ABB RAPID module: P707.mod

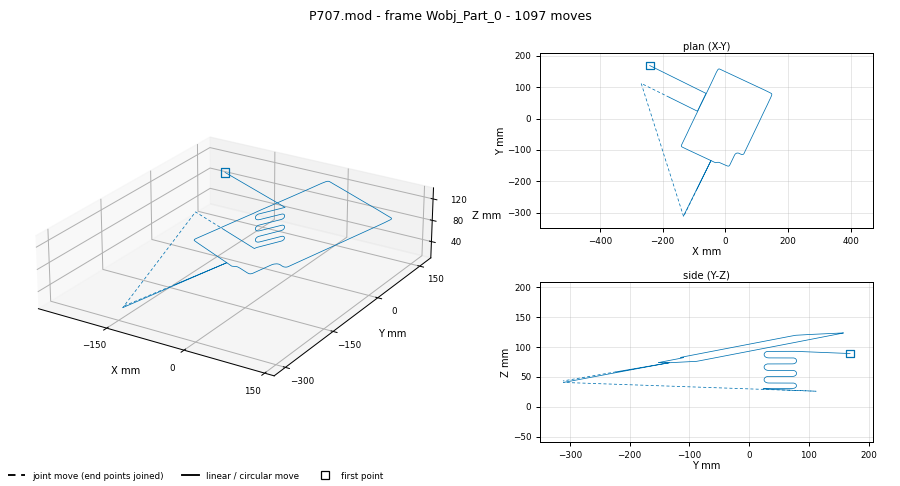
[picture p0: tool path of P707.mod in frame Wobj_Part_0, 1097 of 1107 moves have a stored position in this frame; points joined in program order, loops and branches not executed]
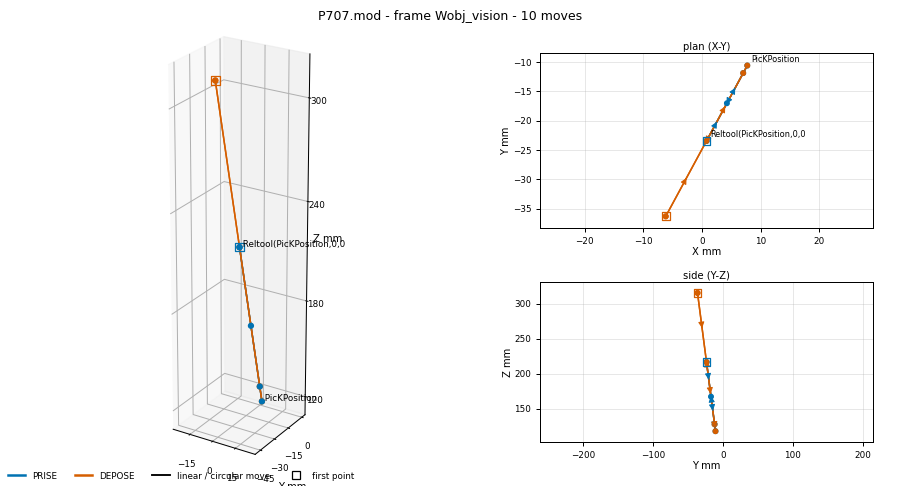
[picture p1: tool path of P707.mod in frame Wobj_vision, 10 of 1107 moves have a stored position in this frame; points joined in program order, loops and branches not executed]
MODULE P707

    ! Nom         :P707
    ! Description :
    ! Créé le     :30/05/2023 16:24:55

    LOCAL CONST SPEEDDATA VitesseLente :=[3,500,0,0];
	LOCAL CONST SPEEDDATA VitesseRapide :=[30,500,0,0];
	LOCAL CONST SPEEDDATA VitesseTronconnage :=[2,500,0,0];
	LOCAL CONST SPEEDDATA VitesseTronconnageApp :=[10,500,0,0];
    !
    !Point de prise
    LOCAL PERS Robtarget PicKPosition := [[7.7250060607796,-10.5869305006045,117.632375104374],[0.0368021435703274,-0.850900226645692,-0.520193892005484,-0.0633460436264631],[0,0,0,0],[8.999999E+09,8.999999E+09,8.999999E+09,8.999999E+09,8.999999E+09,8.999999E+09]];
	LOCAL PERS Pose Ref := [[0,0,0],[1,0,0,0]];
    !
    !Declaration des points de meulage

    !Tr_meulage_motif_1 : Meulage d'un motif
    LOCAL CONST Robtarget Tr_meulage_motif_1_0 := [[-61.692015625,80.0117578125,92.8283359375],[0.376363228761976,-0.369466106511504,0.595187364718739,-0.60629820802494],[0,0,0,0],[8.999999E+09,8.999999E+09,8.999999E+09,8.999999E+09,8.999999E+09,8.999999E+09]];
    LOCAL CONST Robtarget Tr_meulage_motif_1_1 := [[-62.12769921875,79.11165625,92.8283359375],[0.376363228761976,-0.369466106511504,0.595187364718739,-0.60629820802494],[0,0,0,0],[8.999999E+09,8.999999E+09,8.999999E+09,8.999999E+09,8.999999E+09,8.999999E+09]];
    LOCAL CONST Robtarget Tr_meulage_motif_1_2 := [[-62.5633828125,78.2115546875,92.82834375],[0.376363228761976,-0.369466106511504,0.595187364718739,-0.60629820802494],[0,0,0,0],[8.999999E+09,8.999999E+09,8.999999E+09,8.999999E+09,8.999999E+09,8.999999E+09]];
    LOCAL CONST Robtarget Tr_meulage_motif_1_3 := [[-62.99906640625,77.3114609375,92.82834375],[0.376363228761976,-0.369466106511504,0.595187364718739,-0.60629820802494],[0,0,0,0],[8.999999E+09,8.999999E+09,8.999999E+09,8.999999E+09,8.999999E+09,8.999999E+09]];
    LOCAL CONST Robtarget Tr_meulage_motif_1_4 := [[-63.43475,76.411359375,92.8283515625],[0.376363228761976,-0.369466106511504,0.595187364718739,-0.60629820802494],[0,0,0,0],[8.999999E+09,8.999999E+09,8.999999E+09,8.999999E+09,8.999999E+09,8.999999E+09]];
    LOCAL CONST Robtarget Tr_meulage_motif_1_5 := [[-63.8704375,75.5112578125,92.8283515625],[0.376363228761976,-0.369466106511504,0.595187364718739,-0.60629820802494],[0,0,0,0],[8.999999E+09,8.999999E+09,8.999999E+09,8.999999E+09,8.999999E+09,8.999999E+09]];
    LOCAL CONST Robtarget Tr_meulage_motif_1_6 := [[-64.30612109375,74.61115625,92.828359375],[0.376363228761976,-0.369466106511504,0.595187364718739,-0.60629820802494],[0,0,0,0],[8.999999E+09,8.999999E+09,8.999999E+09,8.999999E+09,8.999999E+09,8.999999E+09]];
    LOCAL CONST Robtarget Tr_meulage_motif_1_7 := [[-64.7418046875,73.7110625,92.828359375],[0.376363228761976,-0.369466106511504,0.595187364718739,-0.60629820802494],[0,0,0,0],[8.999999E+09,8.999999E+09,8.999999E+09,8.999999E+09,8.999999E+09,8.999999E+09]];
    LOCAL CONST Robtarget Tr_meulage_motif_1_8 := [[-65.17748828125,72.8109609375,92.828359375],[0.376363228761976,-0.369466106511504,0.595187364718739,-0.60629820802494],[0,0,0,0],[8.999999E+09,8.999999E+09,8.999999E+09,8.999999E+09,8.999999E+09,8.999999E+09]];
    LOCAL CONST Robtarget Tr_meulage_motif_1_9 := [[-65.613171875,71.910859375,92.8283671875],[0.376363228761976,-0.369466106511504,0.595187364718739,-0.60629820802494],[0,0,0,0],[8.999999E+09,8.999999E+09,8.999999E+09,8.999999E+09,8.999999E+09,8.999999E+09]];
    LOCAL CONST Robtarget Tr_meulage_motif_1_10 := [[-66.048859375,71.0107578125,92.8283671875],[0.376363228761976,-0.369466106511504,0.595187364718739,-0.60629820802494],[0,0,0,0],[8.999999E+09,8.999999E+09,8.999999E+09,8.999999E+09,8.999999E+09,8.999999E+09]];
    LOCAL CONST Robtarget Tr_meulage_motif_1_11 := [[-66.4845390625,70.1106640625,92.828375],[0.376363228761976,-0.369466106511504,0.595187364718739,-0.60629820802494],[0,0,0,0],[8.999999E+09,8.999999E+09,8.999999E+09,8.999999E+09,8.999999E+09,8.999999E+09]];
    LOCAL CONST Robtarget Tr_meulage_motif_1_12 := [[-66.9202265625,69.2105625,92.828375],[0.376363228761976,-0.369466106511504,0.595187364718739,-0.60629820802494],[0,0,0,0],[8.999999E+09,8.999999E+09,8.999999E+09,8.999999E+09,8.999999E+09,8.999999E+09]];
    LOCAL CONST Robtarget Tr_meulage_motif_1_13 := [[-67.35590625,68.3104609375,92.8283828125],[0.376363228761976,-0.369466106511504,0.595187364718739,-0.60629820802494],[0,0,0,0],[8.999999E+09,8.999999E+09,8.999999E+09,8.999999E+09,8.999999E+09,8.999999E+09]];
    LOCAL CONST Robtarget Tr_meulage_motif_1_14 := [[-67.79159375,67.410359375,92.8283828125],[0.376363228761976,-0.369466106511504,0.595187364718739,-0.60629820802494],[0,0,0,0],[8.999999E+09,8.999999E+09,8.999999E+09,8.999999E+09,8.999999E+09,8.999999E+09]];
    LOCAL CONST Robtarget Tr_meulage_motif_1_15 := [[-68.22728125,66.510265625,92.8283828125],[0.376363228761976,-0.369466106511504,0.595187364718739,-0.60629820802494],[0,0,0,0],[8.999999E+09,8.999999E+09,8.999999E+09,8.999999E+09,8.999999E+09,8.999999E+09]];
    LOCAL CONST Robtarget Tr_meulage_motif_1_16 := [[-68.6629609375,65.6101640625,92.828390625],[0.376363228761976,-0.369466106511504,0.595187364718739,-0.60629820802494],[0,0,0,0],[8.999999E+09,8.999999E+09,8.999999E+09,8.999999E+09,8.999999E+09,8.999999E+09]];
    LOCAL CONST Robtarget Tr_meulage_motif_1_17 := [[-69.0986484375,64.7100625,92.828390625],[0.376363228761976,-0.369466106511504,0.595187364718739,-0.60629820802494],[0,0,0,0],[8.999999E+09,8.999999E+09,8.999999E+09,8.999999E+09,8.999999E+09,8.999999E+09]];
    LOCAL CONST Robtarget Tr_meulage_motif_1_18 := [[-69.534328125,63.80996484375,92.8283984375],[0.376363228761976,-0.369466106511504,0.595187364718739,-0.60629820802494],[0,0,0,0],[8.999999E+09,8.999999E+09,8.999999E+09,8.999999E+09,8.999999E+09,8.999999E+09]];
    LOCAL CONST Robtarget Tr_meulage_motif_1_19 := [[-69.970015625,62.90986328125,92.8283984375],[0.376363228761976,-0.369466106511504,0.595187364718739,-0.60629820802494],[0,0,0,0],[8.999999E+09,8.999999E+09,8.999999E+09,8.999999E+09,8.999999E+09,8.999999E+09]];
    LOCAL CONST Robtarget Tr_meulage_motif_1_20 := [[-70.405703125,62.009765625,92.82840625],[0.376363228761976,-0.369466106511504,0.595187364718739,-0.60629820802494],[0,0,0,0],[8.999999E+09,8.999999E+09,8.999999E+09,8.999999E+09,8.999999E+09,8.999999E+09]];
    LOCAL CONST Robtarget Tr_meulage_motif_1_21 := [[-70.8413828125,61.1096640625,92.82840625],[0.376363228761976,-0.369466106511504,0.595187364718739,-0.60629820802494],[0,0,0,0],[8.999999E+09,8.999999E+09,8.999999E+09,8.999999E+09,8.999999E+09,8.999999E+09]];
    LOCAL CONST Robtarget Tr_meulage_motif_1_22 := [[-71.2770703125,60.20956640625,92.82840625],[0.376363228761976,-0.369466106511504,0.595187364718739,-0.60629820802494],[0,0,0,0],[8.999999E+09,8.999999E+09,8.999999E+09,8.999999E+09,8.999999E+09,8.999999E+09]];
    LOCAL CONST Robtarget Tr_meulage_motif_1_23 := [[-71.71275,59.30946484375,92.8284140625],[0.376363228761976,-0.369466106511504,0.595187364718739,-0.60629820802494],[0,0,0,0],[8.999999E+09,8.999999E+09,8.999999E+09,8.999999E+09,8.999999E+09,8.999999E+09]];
    LOCAL CONST Robtarget Tr_meulage_motif_1_24 := [[-72.1484375,58.4093671875,92.8284140625],[0.376363228761976,-0.369466106511504,0.595187364718739,-0.60629820802494],[0,0,0,0],[8.999999E+09,8.999999E+09,8.999999E+09,8.999999E+09,8.999999E+09,8.999999E+09]];
    LOCAL CONST Robtarget Tr_meulage_motif_1_25 := [[-72.5841171875,57.509265625,92.828421875],[0.376363228761976,-0.369466106511504,0.595187364718739,-0.60629820802494],[0,0,0,0],[8.999999E+09,8.999999E+09,8.999999E+09,8.999999E+09,8.999999E+09,8.999999E+09]];
    LOCAL CONST Robtarget Tr_meulage_motif_1_26 := [[-73.0198046875,56.60916796875,92.828421875],[0.376363228761976,-0.369466106511504,0.595187364718739,-0.60629820802494],[0,0,0,0],[8.999999E+09,8.999999E+09,8.999999E+09,8.999999E+09,8.999999E+09,8.999999E+09]];
    LOCAL CONST Robtarget Tr_meulage_motif_1_27 := [[-73.4554921875,55.70906640625,92.8284296875],[0.376363228761976,-0.369466106511504,0.595187364718739,-0.60629820802494],[0,0,0,0],[8.999999E+09,8.999999E+09,8.999999E+09,8.999999E+09,8.999999E+09,8.999999E+09]];
    LOCAL CONST Robtarget Tr_meulage_motif_1_28 := [[-73.891171875,54.80896875,92.8284296875],[0.376363228761976,-0.369466106511504,0.595187364718739,-0.60629820802494],[0,0,0,0],[8.999999E+09,8.999999E+09,8.999999E+09,8.999999E+09,8.999999E+09,8.999999E+09]];
    LOCAL CONST Robtarget Tr_meulage_motif_1_29 := [[-74.326859375,53.9088671875,92.8284296875],[0.376363228761976,-0.369466106511504,0.595187364718739,-0.60629820802494],[0,0,0,0],[8.999999E+09,8.999999E+09,8.999999E+09,8.999999E+09,8.999999E+09,8.999999E+09]];
    LOCAL CONST Robtarget Tr_meulage_motif_1_30 := [[-74.7625390625,53.00876953125,92.8284375],[0.376363228761976,-0.369466106511504,0.595187364718739,-0.60629820802494],[0,0,0,0],[8.999999E+09,8.999999E+09,8.999999E+09,8.999999E+09,8.999999E+09,8.999999E+09]];
    LOCAL CONST Robtarget Tr_meulage_motif_1_31 := [[-75.1982265625,52.10866796875,92.8284375],[0.376363228761976,-0.369466106511504,0.595187364718739,-0.60629820802494],[0,0,0,0],[8.999999E+09,8.999999E+09,8.999999E+09,8.999999E+09,8.999999E+09,8.999999E+09]];
    LOCAL CONST Robtarget Tr_meulage_motif_1_32 := [[-75.6339140625,51.2085703125,92.8284453125],[0.376363228761976,-0.369466106511504,0.595187364718739,-0.60629820802494],[0,0,0,0],[8.999999E+09,8.999999E+09,8.999999E+09,8.999999E+09,8.999999E+09,8.999999E+09]];
    LOCAL CONST Robtarget Tr_meulage_motif_1_33 := [[-76.06959375,50.30846875,92.8284453125],[0.376363228761976,-0.369466106511504,0.595187364718739,-0.60629820802494],[0,0,0,0],[8.999999E+09,8.999999E+09,8.999999E+09,8.999999E+09,8.999999E+09,8.999999E+09]];
    LOCAL CONST Robtarget Tr_meulage_motif_1_34 := [[-76.50528125,49.40837109375,92.828453125],[0.376363228761976,-0.369466106511504,0.595187364718739,-0.60629820802494],[0,0,0,0],[8.999999E+09,8.999999E+09,8.999999E+09,8.999999E+09,8.999999E+09,8.999999E+09]];
    LOCAL CONST Robtarget Tr_meulage_motif_1_35 := [[-76.9409609375,48.50826953125,92.828453125],[0.376363228761976,-0.369466106511504,0.595187364718739,-0.60629820802494],[0,0,0,0],[8.999999E+09,8.999999E+09,8.999999E+09,8.999999E+09,8.999999E+09,8.999999E+09]];
    LOCAL CONST Robtarget Tr_meulage_motif_1_36 := [[-77.3766484375,47.608171875,92.828453125],[0.376363228761976,-0.369466106511504,0.595187364718739,-0.60629820802494],[0,0,0,0],[8.999999E+09,8.999999E+09,8.999999E+09,8.999999E+09,8.999999E+09,8.999999E+09]];
    LOCAL CONST Robtarget Tr_meulage_motif_1_37 := [[-77.812328125,46.7080703125,92.8284609375],[0.376363228761976,-0.369466106511504,0.595187364718739,-0.60629820802494],[0,0,0,0],[8.999999E+09,8.999999E+09,8.999999E+09,8.999999E+09,8.999999E+09,8.999999E+09]];
    LOCAL CONST Robtarget Tr_meulage_motif_1_38 := [[-78.248015625,45.80797265625,92.8284609375],[0.376363228761976,-0.369466106511504,0.595187364718739,-0.60629820802494],[0,0,0,0],[8.999999E+09,8.999999E+09,8.999999E+09,8.999999E+09,8.999999E+09,8.999999E+09]];
    LOCAL CONST Robtarget Tr_meulage_motif_1_39 := [[-78.683703125,44.907875,92.82846875],[0.376363228761976,-0.369466106511504,0.595187364718739,-0.60629820802494],[0,0,0,0],[8.999999E+09,8.999999E+09,8.999999E+09,8.999999E+09,8.999999E+09,8.999999E+09]];
    LOCAL CONST Robtarget Tr_meulage_motif_1_40 := [[-79.1193828125,44.0077734375,92.82846875],[0.376363228761976,-0.369466106511504,0.595187364718739,-0.60629820802494],[0,0,0,0],[8.999999E+09,8.999999E+09,8.999999E+09,8.999999E+09,8.999999E+09,8.999999E+09]];
    LOCAL CONST Robtarget Tr_meulage_motif_1_41 := [[-79.5550703125,43.10767578125,92.8284765625],[0.376363228761976,-0.369466106511504,0.595187364718739,-0.60629820802494],[0,0,0,0],[8.999999E+09,8.999999E+09,8.999999E+09,8.999999E+09,8.999999E+09,8.999999E+09]];
    LOCAL CONST Robtarget Tr_meulage_motif_1_42 := [[-79.99075,42.20757421875,92.8284765625],[0.376363228761976,-0.369466106511504,0.595187364718739,-0.60629820802494],[0,0,0,0],[8.999999E+09,8.999999E+09,8.999999E+09,8.999999E+09,8.999999E+09,8.999999E+09]];
    LOCAL CONST Robtarget Tr_meulage_motif_1_43 := [[-80.4264375,41.3074765625,92.8284765625],[0.376363228761976,-0.369466106511504,0.595187364718739,-0.60629820802494],[0,0,0,0],[8.999999E+09,8.999999E+09,8.999999E+09,8.999999E+09,8.999999E+09,8.999999E+09]];
    LOCAL CONST Robtarget Tr_meulage_motif_1_44 := [[-80.862125,40.407375,92.828484375],[0.376363228761976,-0.369466106511504,0.595187364718739,-0.60629820802494],[0,0,0,0],[8.999999E+09,8.999999E+09,8.999999E+09,8.999999E+09,8.999999E+09,8.999999E+09]];
    LOCAL CONST Robtarget Tr_meulage_motif_1_45 := [[-81.2978046875,39.50727734375,92.828484375],[0.376363228761976,-0.369466106511504,0.595187364718739,-0.60629820802494],[0,0,0,0],[8.999999E+09,8.999999E+09,8.999999E+09,8.999999E+09,8.999999E+09,8.999999E+09]];
    LOCAL CONST Robtarget Tr_meulage_motif_1_46 := [[-81.7334921875,38.60717578125,92.8284921875],[0.376363228761976,-0.369466106511504,0.595187364718739,-0.60629820802494],[0,0,0,0],[8.999999E+09,8.999999E+09,8.999999E+09,8.999999E+09,8.999999E+09,8.999999E+09]];
    LOCAL CONST Robtarget Tr_meulage_motif_1_47 := [[-82.169171875,37.707078125,92.8284921875],[0.376363228761976,-0.369466106511504,0.595187364718739,-0.60629820802494],[0,0,0,0],[8.999999E+09,8.999999E+09,8.999999E+09,8.999999E+09,8.999999E+09,8.999999E+09]];
    LOCAL CONST Robtarget Tr_meulage_motif_1_48 := [[-82.604859375,36.8069765625,92.8285],[0.376363228761976,-0.369466106511504,0.595187364718739,-0.60629820802494],[0,0,0,0],[8.999999E+09,8.999999E+09,8.999999E+09,8.999999E+09,8.999999E+09,8.999999E+09]];
    LOCAL CONST Robtarget Tr_meulage_motif_1_49 := [[-83.0405390625,35.90687890625,92.8285],[0.376363228761976,-0.369466106511504,0.595187364718739,-0.60629820802494],[0,0,0,0],[8.999999E+09,8.999999E+09,8.999999E+09,8.999999E+09,8.999999E+09,8.999999E+09]];
    LOCAL CONST Robtarget Tr_meulage_motif_1_50 := [[-83.4762265625,35.00677734375,92.8285],[0.376363228761976,-0.369466106511504,0.595187364718739,-0.60629820802494],[0,0,0,0],[8.999999E+09,8.999999E+09,8.999999E+09,8.999999E+09,8.999999E+09,8.999999E+09]];
    LOCAL CONST Robtarget Tr_meulage_motif_1_51 := [[-83.9119140625,34.1066796875,92.8285078125],[0.376363228761976,-0.369466106511504,0.595187364718739,-0.60629820802494],[0,0,0,0],[8.999999E+09,8.999999E+09,8.999999E+09,8.999999E+09,8.999999E+09,8.999999E+09]];
    LOCAL CONST Robtarget Tr_meulage_motif_1_52 := [[-84.34759375,33.206578125,92.8285078125],[0.376363228761976,-0.369466106511504,0.595187364718739,-0.60629820802494],[0,0,0,0],[8.999999E+09,8.999999E+09,8.999999E+09,8.999999E+09,8.999999E+09,8.999999E+09]];
    LOCAL CONST Robtarget Tr_meulage_motif_1_53 := [[-84.78328125,32.306478515625,92.828515625],[0.376363228761976,-0.369466106511504,0.595187364718739,-0.60629820802494],[0,0,0,0],[8.999999E+09,8.999999E+09,8.999999E+09,8.999999E+09,8.999999E+09,8.999999E+09]];
    LOCAL CONST Robtarget Tr_meulage_motif_1_54 := [[-85.2189609375,31.40637890625,92.828515625],[0.376363228761976,-0.369466106511504,0.595187364718739,-0.60629820802494],[0,0,0,0],[8.999999E+09,8.999999E+09,8.999999E+09,8.999999E+09,8.999999E+09,8.999999E+09]];
    LOCAL CONST Robtarget Tr_meulage_motif_1_55 := [[-85.650984375,30.512767578125,92.7179296875],[0.376363228761976,-0.369466106511504,0.595187364718739,-0.60629820802494],[0,0,0,0],[8.999999E+09,8.999999E+09,8.999999E+09,8.999999E+09,8.999999E+09,8.999999E+09]];
    LOCAL CONST Robtarget Tr_meulage_motif_1_56 := [[-86.0625390625,29.660427734375,92.5067421875],[0.376363228761976,-0.369466106511504,0.595187364718739,-0.60629820802494],[0,0,0,0],[8.999999E+09,8.999999E+09,8.999999E+09,8.999999E+09,8.999999E+09,8.999999E+09]];
    LOCAL CONST Robtarget Tr_meulage_motif_1_57 := [[-86.4330078125,28.892388671875,92.23490625],[0.376363228761976,-0.369466106511504,0.595187364718739,-0.60629820802494],[0,0,0,0],[8.999999E+09,8.999999E+09,8.999999E+09,8.999999E+09,8.999999E+09,8.999999E+09]];
    LOCAL CONST Robtarget Tr_meulage_motif_1_58 := [[-86.7586796875,28.216853515625,91.9589765625],[0.376363228761976,-0.369466106511504,0.595187364718739,-0.60629820802494],[0,0,0,0],[8.999999E+09,8.999999E+09,8.999999E+09,8.999999E+09,8.999999E+09,8.999999E+09]];
    LOCAL CONST Robtarget Tr_meulage_motif_1_59 := [[-87.2360234375,27.22463671875,91.342859375],[0.376363228761976,-0.369466106511504,0.595187364718739,-0.60629820802494],[0,0,0,0],[8.999999E+09,8.999999E+09,8.999999E+09,8.999999E+09,8.999999E+09,8.999999E+09]];
    LOCAL CONST Robtarget Tr_meulage_motif_1_60 := [[-87.67884375,26.3014609375,90.4952109375],[0.376363228761976,-0.369466106511504,0.595187364718739,-0.60629820802494],[0,0,0,0],[8.999999E+09,8.999999E+09,8.999999E+09,8.999999E+09,8.999999E+09,8.999999E+09]];
    LOCAL CONST Robtarget Tr_meulage_motif_1_61 := [[-88.044203125,25.536572265625,89.4713515625],[0.376363228761976,-0.369466106511504,0.595187364718739,-0.60629820802494],[0,0,0,0],[8.999999E+09,8.999999E+09,8.999999E+09,8.999999E+09,8.999999E+09,8.999999E+09]];
    LOCAL CONST Robtarget Tr_meulage_motif_1_62 := [[-88.2525859375,25.095095703125,88.355171875],[0.376363228761976,-0.369466106511504,0.595187364718739,-0.60629820802494],[0,0,0,0],[8.999999E+09,8.999999E+09,8.999999E+09,8.999999E+09,8.999999E+09,8.999999E+09]];
    LOCAL CONST Robtarget Tr_meulage_motif_1_63 := [[-88.2616875,25.069435546875,87.6592109375],[0.376363228761976,-0.369466106511504,0.595187364718739,-0.60629820802494],[0,0,0,0],[8.999999E+09,8.999999E+09,8.999999E+09,8.999999E+09,8.999999E+09,8.999999E+09]];
    LOCAL CONST Robtarget Tr_meulage_motif_1_64 := [[-88.259140625,25.06819921875,86.99796875],[0.376363228761976,-0.369466106511504,0.595187364718739,-0.60629820802494],[0,0,0,0],[8.999999E+09,8.999999E+09,8.999999E+09,8.999999E+09,8.999999E+09,8.999999E+09]];
    LOCAL CONST Robtarget Tr_meulage_motif_1_65 := [[-88.2326796875,25.11635546875,86.3368828125],[0.376363228761976,-0.369466106511504,0.595187364718739,-0.60629820802494],[0,0,0,0],[8.999999E+09,8.999999E+09,8.999999E+09,8.999999E+09,8.999999E+09,8.999999E+09]];
    LOCAL CONST Robtarget Tr_meulage_motif_1_66 := [[-88.0113671875,25.5627421875,85.235140625],[0.376363228761976,-0.369466106511504,0.595187364718739,-0.60629820802494],[0,0,0,0],[8.999999E+09,8.999999E+09,8.999999E+09,8.999999E+09,8.999999E+09,8.999999E+09]];
    LOCAL CONST Robtarget Tr_meulage_motif_1_67 := [[-87.6342734375,26.33190625,84.2285234375],[0.376363228761976,-0.369466106511504,0.595187364718739,-0.60629820802494],[0,0,0,0],[8.999999E+09,8.999999E+09,8.999999E+09,8.999999E+09,8.999999E+09,8.999999E+09]];
    LOCAL CONST Robtarget Tr_meulage_motif_1_68 := [[-87.1851953125,27.251525390625,83.3996484375],[0.376363228761976,-0.369466106511504,0.595187364718739,-0.60629820802494],[0,0,0,0],[8.999999E+09,8.999999E+09,8.999999E+09,8.999999E+09,8.999999E+09,8.999999E+09]];
    LOCAL CONST Robtarget Tr_meulage_motif_1_69 := [[-86.8843125,27.86923828125,83.0038984375],[0.376363228761976,-0.369466106511504,0.595187364718739,-0.60629820802494],[0,0,0,0],[8.999999E+09,8.999999E+09,8.999999E+09,8.999999E+09,8.999999E+09,8.999999E+09]];
    LOCAL CONST Robtarget Tr_meulage_motif_1_70 := [[-86.37784375,28.91078125,82.5163671875],[0.376363228761976,-0.369466106511504,0.595187364718739,-0.60629820802494],[0,0,0,0],[8.999999E+09,8.999999E+09,8.999999E+09,8.999999E+09,8.999999E+09,8.999999E+09]];
    LOCAL CONST Robtarget Tr_meulage_motif_1_71 := [[-86.00865625,29.670900390625,82.2522734375],[0.376363228761976,-0.369466106511504,0.595187364718739,-0.60629820802494],[0,0,0,0],[8.999999E+09,8.999999E+09,8.999999E+09,8.999999E+09,8.999999E+09,8.999999E+09]];
    LOCAL CONST Robtarget Tr_meulage_motif_1_72 := [[-85.6018125,30.50941015625,82.0478046875],[0.376363228761976,-0.369466106511504,0.595187364718739,-0.60629820802494],[0,0,0,0],[8.999999E+09,8.999999E+09,8.999999E+09,8.999999E+09,8.999999E+09,8.999999E+09]];
    LOCAL CONST Robtarget Tr_meulage_motif_1_73 := [[-85.1737421875,31.3927109375,81.9392109375],[0.376363228761976,-0.369466106511504,0.595187364718739,-0.60629820802494],[0,0,0,0],[8.999999E+09,8.999999E+09,8.999999E+09,8.999999E+09,8.999999E+09,8.999999E+09]];
    LOCAL CONST Robtarget Tr_meulage_motif_1_74 := [[-84.7408671875,32.28591015625,81.8286171875],[0.376363228761976,-0.369466106511504,0.595187364718739,-0.60629820802494],[0,0,0,0],[8.999999E+09,8.999999E+09,8.999999E+09,8.999999E+09,8.999999E+09,8.999999E+09]];
    LOCAL CONST Robtarget Tr_meulage_motif_1_75 := [[-84.3051875,33.1860078125,81.828609375],[0.376363228761976,-0.369466106511504,0.595187364718739,-0.60629820802494],[0,0,0,0],[8.999999E+09,8.999999E+09,8.999999E+09,8.999999E+09,8.999999E+09,8.999999E+09]];
    LOCAL CONST Robtarget Tr_meulage_motif_1_76 := [[-83.8695,34.086109375,81.828609375],[0.376363228761976,-0.369466106511504,0.595187364718739,-0.60629820802494],[0,0,0,0],[8.999999E+09,8.999999E+09,8.999999E+09,8.999999E+09,8.999999E+09,8.999999E+09]];
    LOCAL CONST Robtarget Tr_meulage_motif_1_77 := [[-83.4338125,34.98620703125,81.8286015625],[0.376363228761976,-0.369466106511504,0.595187364718739,-0.60629820802494],[0,0,0,0],[8.999999E+09,8.999999E+09,8.999999E+09,8.999999E+09,8.999999E+09,8.999999E+09]];
    LOCAL CONST Robtarget Tr_meulage_motif_1_78 := [[-82.9981328125,35.88630859375,81.8286015625],[0.376363228761976,-0.369466106511504,0.595187364718739,-0.60629820802494],[0,0,0,0],[8.999999E+09,8.999999E+09,8.999999E+09,8.999999E+09,8.999999E+09,8.999999E+09]];
    LOCAL CONST Robtarget Tr_meulage_motif_1_79 := [[-82.5624453125,36.78640625,81.82859375],[0.376363228761976,-0.369466106511504,0.595187364718739,-0.60629820802494],[0,0,0,0],[8.999999E+09,8.999999E+09,8.999999E+09,8.999999E+09,8.999999E+09,8.999999E+09]];
    LOCAL CONST Robtarget Tr_meulage_motif_1_80 := [[-82.126765625,37.6865078125,81.82859375],[0.376363228761976,-0.369466106511504,0.595187364718739,-0.60629820802494],[0,0,0,0],[8.999999E+09,8.999999E+09,8.999999E+09,8.999999E+09,8.999999E+09,8.999999E+09]];
    LOCAL CONST Robtarget Tr_meulage_motif_1_81 := [[-81.691078125,38.58660546875,81.82859375],[0.376363228761976,-0.369466106511504,0.595187364718739,-0.60629820802494],[0,0,0,0],[8.999999E+09,8.999999E+09,8.999999E+09,8.999999E+09,8.999999E+09,8.999999E+09]];
    LOCAL CONST Robtarget Tr_meulage_motif_1_82 := [[-81.2553984375,39.48670703125,81.8285859375],[0.376363228761976,-0.369466106511504,0.595187364718739,-0.60629820802494],[0,0,0,0],[8.999999E+09,8.999999E+09,8.999999E+09,8.999999E+09,8.999999E+09,8.999999E+09]];
    LOCAL CONST Robtarget Tr_meulage_motif_1_83 := [[-80.8197109375,40.3868046875,81.8285859375],[0.376363228761976,-0.369466106511504,0.595187364718739,-0.60629820802494],[0,0,0,0],[8.999999E+09,8.999999E+09,8.999999E+09,8.999999E+09,8.999999E+09,8.999999E+09]];
    LOCAL CONST Robtarget Tr_meulage_motif_1_84 := [[-80.3840234375,41.28690625,81.828578125],[0.376363228761976,-0.369466106511504,0.595187364718739,-0.60629820802494],[0,0,0,0],[8.999999E+09,8.999999E+09,8.999999E+09,8.999999E+09,8.999999E+09,8.999999E+09]];
    LOCAL CONST Robtarget Tr_meulage_motif_1_85 := [[-79.94834375,42.18700390625,81.828578125],[0.376363228761976,-0.369466106511504,0.595187364718739,-0.60629820802494],[0,0,0,0],[8.999999E+09,8.999999E+09,8.999999E+09,8.999999E+09,8.999999E+09,8.999999E+09]];
    LOCAL CONST Robtarget Tr_meulage_motif_1_86 := [[-79.51265625,43.08710546875,81.8285703125],[0.376363228761976,-0.369466106511504,0.595187364718739,-0.60629820802494],[0,0,0,0],[8.999999E+09,8.999999E+09,8.999999E+09,8.999999E+09,8.999999E+09,8.999999E+09]];
    LOCAL CONST Robtarget Tr_meulage_motif_1_87 := [[-79.0769765625,43.987203125,81.8285703125],[0.376363228761976,-0.369466106511504,0.595187364718739,-0.60629820802494],[0,0,0,0],[8.999999E+09,8.999999E+09,8.999999E+09,8.999999E+09,8.999999E+09,8.999999E+09]];
    LOCAL CONST Robtarget Tr_meulage_motif_1_88 := [[-78.6412890625,44.8873046875,81.8285703125],[0.376363228761976,-0.369466106511504,0.595187364718739,-0.60629820802494],[0,0,0,0],[8.999999E+09,8.999999E+09,8.999999E+09,8.999999E+09,8.999999E+09,8.999999E+09]];
    LOCAL CONST Robtarget Tr_meulage_motif_1_89 := [[-78.2056015625,45.78740234375,81.8285625],[0.376363228761976,-0.369466106511504,0.595187364718739,-0.60629820802494],[0,0,0,0],[8.999999E+09,8.999999E+09,8.999999E+09,8.999999E+09,8.999999E+09,8.999999E+09]];
    LOCAL CONST Robtarget Tr_meulage_motif_1_90 := [[-77.769921875,46.68750390625,81.8285625],[0.376363228761976,-0.369466106511504,0.595187364718739,-0.60629820802494],[0,0,0,0],[8.999999E+09,8.999999E+09,8.999999E+09,8.999999E+09,8.999999E+09,8.999999E+09]];
    LOCAL CONST Robtarget Tr_meulage_motif_1_91 := [[-77.334234375,47.5876015625,81.8285546875],[0.376363228761976,-0.369466106511504,0.595187364718739,-0.60629820802494],[0,0,0,0],[8.999999E+09,8.999999E+09,8.999999E+09,8.999999E+09,8.999999E+09,8.999999E+09]];
    LOCAL CONST Robtarget Tr_meulage_motif_1_92 := [[-76.8985546875,48.487703125,81.8285546875],[0.376363228761976,-0.369466106511504,0.595187364718739,-0.60629820802494],[0,0,0,0],[8.999999E+09,8.999999E+09,8.999999E+09,8.999999E+09,8.999999E+09,8.999999E+09]];
    LOCAL CONST Robtarget Tr_meulage_motif_1_93 := [[-76.4628671875,49.38780078125,81.828546875],[0.376363228761976,-0.369466106511504,0.595187364718739,-0.60629820802494],[0,0,0,0],[8.999999E+09,8.999999E+09,8.999999E+09,8.999999E+09,8.999999E+09,8.999999E+09]];
    LOCAL CONST Robtarget Tr_meulage_motif_1_94 := [[-76.0271875,50.28790234375,81.828546875],[0.376363228761976,-0.369466106511504,0.595187364718739,-0.60629820802494],[0,0,0,0],[8.999999E+09,8.999999E+09,8.999999E+09,8.999999E+09,8.999999E+09,8.999999E+09]];
    LOCAL CONST Robtarget Tr_meulage_motif_1_95 := [[-75.5915,51.188,81.828546875],[0.376363228761976,-0.369466106511504,0.595187364718739,-0.60629820802494],[0,0,0,0],[8.999999E+09,8.999999E+09,8.999999E+09,8.999999E+09,8.999999E+09,8.999999E+09]];
    LOCAL CONST Robtarget Tr_meulage_motif_1_96 := [[-75.1558125,52.0881015625,81.8285390625],[0.376363228761976,-0.369466106511504,0.595187364718739,-0.60629820802494],[0,0,0,0],[8.999999E+09,8.999999E+09,8.999999E+09,8.999999E+09,8.999999E+09,8.999999E+09]];
    LOCAL CONST Robtarget Tr_meulage_motif_1_97 := [[-74.7201328125,52.98819921875,81.8285390625],[0.376363228761976,-0.369466106511504,0.595187364718739,-0.60629820802494],[0,0,0,0],[8.999999E+09,8.999999E+09,8.999999E+09,8.999999E+09,8.999999E+09,8.999999E+09]];
    LOCAL CONST Robtarget Tr_meulage_motif_1_98 := [[-74.2844453125,53.88830078125,81.82853125],[0.376363228761976,-0.369466106511504,0.595187364718739,-0.60629820802494],[0,0,0,0],[8.999999E+09,8.999999E+09,8.999999E+09,8.999999E+09,8.999999E+09,8.999999E+09]];
    LOCAL CONST Robtarget Tr_meulage_motif_1_99 := [[-73.848765625,54.7883984375,81.82853125],[0.376363228761976,-0.369466106511504,0.595187364718739,-0.60629820802494],[0,0,0,0],[8.999999E+09,8.999999E+09,8.999999E+09,8.999999E+09,8.999999E+09,8.999999E+09]];
    LOCAL CONST Robtarget Tr_meulage_motif_1_100 := [[-73.413078125,55.6885,81.8285234375],[0.376363228761976,-0.369466106511504,0.595187364718739,-0.60629820802494],[0,0,0,0],[8.999999E+09,8.999999E+09,8.999999E+09,8.999999E+09,8.999999E+09,8.999999E+09]];
    LOCAL CONST Robtarget Tr_meulage_motif_1_101 := [[-72.977390625,56.58859765625,81.8285234375],[0.376363228761976,-0.369466106511504,0.595187364718739,-0.60629820802494],[0,0,0,0],[8.999999E+09,8.999999E+09,8.999999E+09,8.999999E+09,8.999999E+09,8.999999E+09]];
    LOCAL CONST Robtarget Tr_meulage_motif_1_102 := [[-72.5417109375,57.48869921875,81.8285234375],[0.376363228761976,-0.369466106511504,0.595187364718739,-0.60629820802494],[0,0,0,0],[8.999999E+09,8.999999E+09,8.999999E+09,8.999999E+09,8.999999E+09,8.999999E+09]];
    LOCAL CONST Robtarget Tr_meulage_motif_1_103 := [[-72.1060234375,58.388796875,81.828515625],[0.376363228761976,-0.369466106511504,0.595187364718739,-0.60629820802494],[0,0,0,0],[8.999999E+09,8.999999E+09,8.999999E+09,8.999999E+09,8.999999E+09,8.999999E+09]];
    LOCAL CONST Robtarget Tr_meulage_motif_1_104 := [[-71.67034375,59.2888984375,81.828515625],[0.376363228761976,-0.369466106511504,0.595187364718739,-0.60629820802494],[0,0,0,0],[8.999999E+09,8.999999E+09,8.999999E+09,8.999999E+09,8.999999E+09,8.999999E+09]];
    LOCAL CONST Robtarget Tr_meulage_motif_1_105 := [[-71.23465625,60.18899609375,81.8285078125],[0.376363228761976,-0.369466106511504,0.595187364718739,-0.60629820802494],[0,0,0,0],[8.999999E+09,8.999999E+09,8.999999E+09,8.999999E+09,8.999999E+09,8.999999E+09]];
    LOCAL CONST Robtarget Tr_meulage_motif_1_106 := [[-70.7989765625,61.08909765625,81.8285078125],[0.376363228761976,-0.369466106511504,0.595187364718739,-0.60629820802494],[0,0,0,0],[8.999999E+09,8.999999E+09,8.999999E+09,8.999999E+09,8.999999E+09,8.999999E+09]];
    LOCAL CONST Robtarget Tr_meulage_motif_1_107 := [[-70.3632890625,61.9891953125,81.8285],[0.376363228761976,-0.369466106511504,0.595187364718739,-0.60629820802494],[0,0,0,0],[8.999999E+09,8.999999E+09,8.999999E+09,8.999999E+09,8.999999E+09,8.999999E+09]];
    LOCAL CONST Robtarget Tr_meulage_motif_1_108 := [[-69.9276015625,62.889296875,81.8285],[0.376363228761976,-0.369466106511504,0.595187364718739,-0.60629820802494],[0,0,0,0],[8.999999E+09,8.999999E+09,8.999999E+09,8.999999E+09,8.999999E+09,8.999999E+09]];
    LOCAL CONST Robtarget Tr_meulage_motif_1_109 := [[-69.491921875,63.78939453125,81.8285],[0.376363228761976,-0.369466106511504,0.595187364718739,-0.60629820802494],[0,0,0,0],[8.999999E+09,8.999999E+09,8.999999E+09,8.999999E+09,8.999999E+09,8.999999E+09]];
    LOCAL CONST Robtarget Tr_meulage_motif_1_110 := [[-69.056234375,64.68949609375,81.8284921875],[0.376363228761976,-0.369466106511504,0.595187364718739,-0.60629820802494],[0,0,0,0],[8.999999E+09,8.999999E+09,8.999999E+09,8.999999E+09,8.999999E+09,8.999999E+09]];
    LOCAL CONST Robtarget Tr_meulage_motif_1_111 := [[-68.6205546875,65.58959375,81.8284921875],[0.376363228761976,-0.369466106511504,0.595187364718739,-0.60629820802494],[0,0,0,0],[8.999999E+09,8.999999E+09,8.999999E+09,8.999999E+09,8.999999E+09,8.999999E+09]];
    LOCAL CONST Robtarget Tr_meulage_motif_1_112 := [[-68.1848671875,66.4896953125,81.828484375],[0.376363228761976,-0.369466106511504,0.595187364718739,-0.60629820802494],[0,0,0,0],[8.999999E+09,8.999999E+09,8.999999E+09,8.999999E+09,8.999999E+09,8.999999E+09]];
    LOCAL CONST Robtarget Tr_meulage_motif_1_113 := [[-67.7491796875,67.3897890625,81.828484375],[0.376363228761976,-0.369466106511504,0.595187364718739,-0.60629820802494],[0,0,0,0],[8.999999E+09,8.999999E+09,8.999999E+09,8.999999E+09,8.999999E+09,8.999999E+09]];
    LOCAL CONST Robtarget Tr_meulage_motif_1_114 := [[-67.3135,68.289890625,81.8284765625],[0.376363228761976,-0.369466106511504,0.595187364718739,-0.60629820802494],[0,0,0,0],[8.999999E+09,8.999999E+09,8.999999E+09,8.999999E+09,8.999999E+09,8.999999E+09]];
    LOCAL CONST Robtarget Tr_meulage_motif_1_115 := [[-66.8778125,69.1899921875,81.8284765625],[0.376363228761976,-0.369466106511504,0.595187364718739,-0.60629820802494],[0,0,0,0],[8.999999E+09,8.999999E+09,8.999999E+09,8.999999E+09,8.999999E+09,8.999999E+09]];
    LOCAL CONST Robtarget Tr_meulage_motif_1_116 := [[-66.4421328125,70.09009375,81.8284765625],[0.376363228761976,-0.369466106511504,0.595187364718739,-0.60629820802494],[0,0,0,0],[8.999999E+09,8.999999E+09,8.999999E+09,8.999999E+09,8.999999E+09,8.999999E+09]];
    LOCAL CONST Robtarget Tr_meulage_motif_1_117 := [[-66.0064453125,70.9901875,81.82846875],[0.376363228761976,-0.369466106511504,0.595187364718739,-0.60629820802494],[0,0,0,0],[8.999999E+09,8.999999E+09,8.999999E+09,8.999999E+09,8.999999E+09,8.999999E+09]];
    LOCAL CONST Robtarget Tr_meulage_motif_1_118 := [[-65.570765625,71.8902890625,81.82846875],[0.376363228761976,-0.369466106511504,0.595187364718739,-0.60629820802494],[0,0,0,0],[8.999999E+09,8.999999E+09,8.999999E+09,8.999999E+09,8.999999E+09,8.999999E+09]];
    LOCAL CONST Robtarget Tr_meulage_motif_1_119 := [[-65.135078125,72.790390625,81.8284609375],[0.376363228761976,-0.369466106511504,0.595187364718739,-0.60629820802494],[0,0,0,0],[8.999999E+09,8.999999E+09,8.999999E+09,8.999999E+09,8.999999E+09,8.999999E+09]];
    LOCAL CONST Robtarget Tr_meulage_motif_1_120 := [[-64.69939453125,73.6904921875,81.8284609375],[0.376363228761976,-0.369466106511504,0.595187364718739,-0.60629820802494],[0,0,0,0],[8.999999E+09,8.999999E+09,8.999999E+09,8.999999E+09,8.999999E+09,8.999999E+09]];
    LOCAL CONST Robtarget Tr_meulage_motif_1_121 := [[-64.2665234375,74.5836875,81.7178671875],[0.376363228761976,-0.369466106511504,0.595187364718739,-0.60629820802494],[0,0,0,0],[8.999999E+09,8.999999E+09,8.999999E+09,8.999999E+09,8.999999E+09,8.999999E+09]];
    LOCAL CONST Robtarget Tr_meulage_motif_1_122 := [[-63.85333203125,75.435234375,81.506671875],[0.376363228761976,-0.369466106511504,0.595187364718739,-0.60629820802494],[0,0,0,0],[8.999999E+09,8.999999E+09,8.999999E+09,8.999999E+09,8.999999E+09,8.999999E+09]];
    LOCAL CONST Robtarget Tr_meulage_motif_1_123 := [[-63.48076953125,76.2022578125,81.234828125],[0.376363228761976,-0.369466106511504,0.595187364718739,-0.60629820802494],[0,0,0,0],[8.999999E+09,8.999999E+09,8.999999E+09,8.999999E+09,8.999999E+09,8.999999E+09]];
    LOCAL CONST Robtarget Tr_meulage_motif_1_124 := [[-63.169609375,76.842109375,80.930671875],[0.376363228761976,-0.369466106511504,0.595187364718739,-0.60629820802494],[0,0,0,0],[8.999999E+09,8.999999E+09,8.999999E+09,8.999999E+09,8.999999E+09,8.999999E+09]];
    LOCAL CONST Robtarget Tr_meulage_motif_1_125 := [[-62.7163515625,77.772,80.2681484375],[0.376363228761976,-0.369466106511504,0.595187364718739,-0.60629820802494],[0,0,0,0],[8.999999E+09,8.999999E+09,8.999999E+09,8.999999E+09,8.999999E+09,8.999999E+09]];
    LOCAL CONST Robtarget Tr_meulage_motif_1_126 := [[-62.3199140625,78.5821484375,79.3662109375],[0.376363228761976,-0.369466106511504,0.595187364718739,-0.60629820802494],[0,0,0,0],[8.999999E+09,8.999999E+09,8.999999E+09,8.999999E+09,8.999999E+09,8.999999E+09]];
    LOCAL CONST Robtarget Tr_meulage_motif_1_127 := [[-62.0828046875,79.06171875,78.3201875],[0.376363228761976,-0.369466106511504,0.595187364718739,-0.60629820802494],[0,0,0,0],[8.999999E+09,8.999999E+09,8.999999E+09,8.999999E+09,8.999999E+09,8.999999E+09]];
    LOCAL CONST Robtarget Tr_meulage_motif_1_128 := [[-61.999625,79.2267421875,77.6269765625],[0.376363228761976,-0.369466106511504,0.595187364718739,-0.60629820802494],[0,0,0,0],[8.999999E+09,8.999999E+09,8.999999E+09,8.999999E+09,8.999999E+09,8.999999E+09]];
    LOCAL CONST Robtarget Tr_meulage_motif_1_129 := [[-61.96883984375,79.282765625,76.856984375],[0.376363228761976,-0.369466106511504,0.595187364718739,-0.60629820802494],[0,0,0,0],[8.999999E+09,8.999999E+09,8.999999E+09,8.999999E+09,8.999999E+09,8.999999E+09]];
    LOCAL CONST Robtarget Tr_meulage_motif_1_130 := [[-61.99503515625,79.221078125,76.0871171875],[0.376363228761976,-0.369466106511504,0.595187364718739,-0.60629820802494],[0,0,0,0],[8.999999E+09,8.999999E+09,8.999999E+09,8.999999E+09,8.999999E+09,8.999999E+09]];
    LOCAL CONST Robtarget Tr_meulage_motif_1_131 := [[-62.17357421875,78.841328125,74.9788828125],[0.376363228761976,-0.369466106511504,0.595187364718739,-0.60629820802494],[0,0,0,0],[8.999999E+09,8.999999E+09,8.999999E+09,8.999999E+09,8.999999E+09,8.999999E+09]];
    LOCAL CONST Robtarget Tr_meulage_motif_1_132 := [[-62.35182421875,78.4673125,74.3931953125],[0.376363228761976,-0.369466106511504,0.595187364718739,-0.60629820802494],[0,0,0,0],[8.999999E+09,8.999999E+09,8.999999E+09,8.999999E+09,8.999999E+09,8.999999E+09]];
    LOCAL CONST Robtarget Tr_meulage_motif_1_133 := [[-62.73491015625,77.6671484375,73.5060859375],[0.376363228761976,-0.369466106511504,0.595187364718739,-0.60629820802494],[0,0,0,0],[8.999999E+09,8.999999E+09,8.999999E+09,8.999999E+09,8.999999E+09,8.999999E+09]];
    LOCAL CONST Robtarget Tr_meulage_motif_1_134 := [[-62.98848828125,77.1391953125,73.09178125],[0.376363228761976,-0.369466106511504,0.595187364718739,-0.60629820802494],[0,0,0,0],[8.999999E+09,8.999999E+09,8.999999E+09,8.999999E+09,8.999999E+09,8.999999E+09]];
    LOCAL CONST Robtarget Tr_meulage_motif_1_135 := [[-63.4734453125,76.131953125,72.5476953125],[0.376363228761976,-0.369466106511504,0.595187364718739,-0.60629820802494],[0,0,0,0],[8.999999E+09,8.999999E+09,8.999999E+09,8.999999E+09,8.999999E+09,8.999999E+09]];
    LOCAL CONST Robtarget Tr_meulage_motif_1_136 := [[-63.83200390625,75.38828125,72.2521953125],[0.376363228761976,-0.369466106511504,0.595187364718739,-0.60629820802494],[0,0,0,0],[8.999999E+09,8.999999E+09,8.999999E+09,8.999999E+09,8.999999E+09,8.999999E+09]];
    LOCAL CONST Robtarget Tr_meulage_motif_1_137 := [[-64.2372734375,74.5490078125,72.047734375],[0.376363228761976,-0.369466106511504,0.595187364718739,-0.60629820802494],[0,0,0,0],[8.999999E+09,8.999999E+09,8.999999E+09,8.999999E+09,8.999999E+09,8.999999E+09]];
    LOCAL CONST Robtarget Tr_meulage_motif_1_138 := [[-64.66450390625,73.6653046875,71.9391484375],[0.376363228761976,-0.369466106511504,0.595187364718739,-0.60629820802494],[0,0,0,0],[8.999999E+09,8.999999E+09,8.999999E+09,8.999999E+09,8.999999E+09,8.999999E+09]];
    LOCAL CONST Robtarget Tr_meulage_motif_1_139 := [[-65.0965234375,72.7716875,71.8285546875],[0.376363228761976,-0.369466106511504,0.595187364718739,-0.60629820802494],[0,0,0,0],[8.999999E+09,8.999999E+09,8.999999E+09,8.999999E+09,8.999999E+09,8.999999E+09]];
    LOCAL CONST Robtarget Tr_meulage_motif_1_140 := [[-65.53220703125,71.87159375,71.8285625],[0.376363228761976,-0.369466106511504,0.595187364718739,-0.60629820802494],[0,0,0,0],[8.999999E+09,8.999999E+09,8.999999E+09,8.999999E+09,8.999999E+09,8.999999E+09]];
    LOCAL CONST Robtarget Tr_meulage_motif_1_141 := [[-65.967890625,70.9714921875,71.8285625],[0.376363228761976,-0.369466106511504,0.595187364718739,-0.60629820802494],[0,0,0,0],[8.999999E+09,8.999999E+09,8.999999E+09,8.999999E+09,8.999999E+09,8.999999E+09]];
    LOCAL CONST Robtarget Tr_meulage_motif_1_142 := [[-66.403578125,70.071390625,71.8285625],[0.376363228761976,-0.369466106511504,0.595187364718739,-0.60629820802494],[0,0,0,0],[8.999999E+09,8.999999E+09,8.999999E+09,8.999999E+09,8.999999E+09,8.999999E+09]];
    LOCAL CONST Robtarget Tr_meulage_motif_1_143 := [[-66.8392578125,69.1712890625,71.8285703125],[0.376363228761976,-0.369466106511504,0.595187364718739,-0.60629820802494],[0,0,0,0],[8.999999E+09,8.999999E+09,8.999999E+09,8.999999E+09,8.999999E+09,8.999999E+09]];
    LOCAL CONST Robtarget Tr_meulage_motif_1_144 := [[-67.2749453125,68.2711953125,71.8285703125],[0.376363228761976,-0.369466106511504,0.595187364718739,-0.60629820802494],[0,0,0,0],[8.999999E+09,8.999999E+09,8.999999E+09,8.999999E+09,8.999999E+09,8.999999E+09]];
    LOCAL CONST Robtarget Tr_meulage_motif_1_145 := [[-67.710625,67.37109375,71.828578125],[0.376363228761976,-0.369466106511504,0.595187364718739,-0.60629820802494],[0,0,0,0],[8.999999E+09,8.999999E+09,8.999999E+09,8.999999E+09,8.999999E+09,8.999999E+09]];
    LOCAL CONST Robtarget Tr_meulage_motif_1_146 := [[-68.1463125,66.4709921875,71.828578125],[0.376363228761976,-0.369466106511504,0.595187364718739,-0.60629820802494],[0,0,0,0],[8.999999E+09,8.999999E+09,8.999999E+09,8.999999E+09,8.999999E+09,8.999999E+09]];
    LOCAL CONST Robtarget Tr_meulage_motif_1_147 := [[-68.582,65.570890625,71.8285859375],[0.376363228761976,-0.369466106511504,0.595187364718739,-0.60629820802494],[0,0,0,0],[8.999999E+09,8.999999E+09,8.999999E+09,8.999999E+09,8.999999E+09,8.999999E+09]];
    LOCAL CONST Robtarget Tr_meulage_motif_1_148 := [[-69.0176796875,64.67079296875,71.8285859375],[0.376363228761976,-0.369466106511504,0.595187364718739,-0.60629820802494],[0,0,0,0],[8.999999E+09,8.999999E+09,8.999999E+09,8.999999E+09,8.999999E+09,8.999999E+09]];
    LOCAL CONST Robtarget Tr_meulage_motif_1_149 := [[-69.4533671875,63.7706953125,71.8285859375],[0.376363228761976,-0.369466106511504,0.595187364718739,-0.60629820802494],[0,0,0,0],[8.999999E+09,8.999999E+09,8.999999E+09,8.999999E+09,8.999999E+09,8.999999E+09]];
    LOCAL CONST Robtarget Tr_meulage_motif_1_150 := [[-69.889046875,62.87059375,71.82859375],[0.376363228761976,-0.369466106511504,0.595187364718739,-0.60629820802494],[0,0,0,0],[8.999999E+09,8.999999E+09,8.999999E+09,8.999999E+09,8.999999E+09,8.999999E+09]];
    LOCAL CONST Robtarget Tr_meulage_motif_1_151 := [[-70.324734375,61.97049609375,71.82859375],[0.376363228761976,-0.369466106511504,0.595187364718739,-0.60629820802494],[0,0,0,0],[8.999999E+09,8.999999E+09,8.999999E+09,8.999999E+09,8.999999E+09,8.999999E+09]];
    LOCAL CONST Robtarget Tr_meulage_motif_1_152 := [[-70.7604140625,61.0703984375,71.8286015625],[0.376363228761976,-0.369466106511504,0.595187364718739,-0.60629820802494],[0,0,0,0],[8.999999E+09,8.999999E+09,8.999999E+09,8.999999E+09,8.999999E+09,8.999999E+09]];
    LOCAL CONST Robtarget Tr_meulage_motif_1_153 := [[-71.1961015625,60.170296875,71.8286015625],[0.376363228761976,-0.369466106511504,0.595187364718739,-0.60629820802494],[0,0,0,0],[8.999999E+09,8.999999E+09,8.999999E+09,8.999999E+09,8.999999E+09,8.999999E+09]];
    LOCAL CONST Robtarget Tr_meulage_motif_1_154 := [[-71.6317890625,59.27019921875,71.828609375],[0.376363228761976,-0.369466106511504,0.595187364718739,-0.60629820802494],[0,0,0,0],[8.999999E+09,8.999999E+09,8.999999E+09,8.999999E+09,8.999999E+09,8.999999E+09]];
    LOCAL CONST Robtarget Tr_meulage_motif_1_155 := [[-72.06746875,58.37009765625,71.828609375],[0.376363228761976,-0.369466106511504,0.595187364718739,-0.60629820802494],[0,0,0,0],[8.999999E+09,8.999999E+09,8.999999E+09,8.999999E+09,8.999999E+09,8.999999E+09]];
    LOCAL CONST Robtarget Tr_meulage_motif_1_156 := [[-72.50315625,57.47,71.828609375],[0.376363228761976,-0.369466106511504,0.595187364718739,-0.60629820802494],[0,0,0,0],[8.999999E+09,8.999999E+09,8.999999E+09,8.999999E+09,8.999999E+09,8.999999E+09]];
    LOCAL CONST Robtarget Tr_meulage_motif_1_157 := [[-72.9388359375,56.5698984375,71.8286171875],[0.376363228761976,-0.369466106511504,0.595187364718739,-0.60629820802494],[0,0,0,0],[8.999999E+09,8.999999E+09,8.999999E+09,8.999999E+09,8.999999E+09,8.999999E+09]];
    LOCAL CONST Robtarget Tr_meulage_motif_1_158 := [[-73.3745234375,55.66980078125,71.8286171875],[0.376363228761976,-0.369466106511504,0.595187364718739,-0.60629820802494],[0,0,0,0],[8.999999E+09,8.999999E+09,8.999999E+09,8.999999E+09,8.999999E+09,8.999999E+09]];
    LOCAL CONST Robtarget Tr_meulage_motif_1_159 := [[-73.8102109375,54.76969921875,71.828625],[0.376363228761976,-0.369466106511504,0.595187364718739,-0.60629820802494],[0,0,0,0],[8.999999E+09,8.999999E+09,8.999999E+09,8.999999E+09,8.999999E+09,8.999999E+09]];
    LOCAL CONST Robtarget Tr_meulage_motif_1_160 := [[-74.245890625,53.8696015625,71.828625],[0.376363228761976,-0.369466106511504,0.595187364718739,-0.60629820802494],[0,0,0,0],[8.999999E+09,8.999999E+09,8.999999E+09,8.999999E+09,8.999999E+09,8.999999E+09]];
    LOCAL CONST Robtarget Tr_meulage_motif_1_161 := [[-74.681578125,52.9695,71.8286328125],[0.376363228761976,-0.369466106511504,0.595187364718739,-0.60629820802494],[0,0,0,0],[8.999999E+09,8.999999E+09,8.999999E+09,8.999999E+09,8.999999E+09,8.999999E+09]];
    LOCAL CONST Robtarget Tr_meulage_motif_1_162 := [[-75.1172578125,52.06940234375,71.8286328125],[0.376363228761976,-0.369466106511504,0.595187364718739,-0.60629820802494],[0,0,0,0],[8.999999E+09,8.999999E+09,8.999999E+09,8.999999E+09,8.999999E+09,8.999999E+09]];
    LOCAL CONST Robtarget Tr_meulage_motif_1_163 := [[-75.5529453125,51.16930078125,71.8286328125],[0.376363228761976,-0.369466106511504,0.595187364718739,-0.60629820802494],[0,0,0,0],[8.999999E+09,8.999999E+09,8.999999E+09,8.999999E+09,8.999999E+09,8.999999E+09]];
    LOCAL CONST Robtarget Tr_meulage_motif_1_164 := [[-75.988625,50.269203125,71.828640625],[0.376363228761976,-0.369466106511504,0.595187364718739,-0.60629820802494],[0,0,0,0],[8.999999E+09,8.999999E+09,8.999999E+09,8.999999E+09,8.999999E+09,8.999999E+09]];
    LOCAL CONST Robtarget Tr_meulage_motif_1_165 := [[-76.4243125,49.3691015625,71.828640625],[0.376363228761976,-0.369466106511504,0.595187364718739,-0.60629820802494],[0,0,0,0],[8.999999E+09,8.999999E+09,8.999999E+09,8.999999E+09,8.999999E+09,8.999999E+09]];
    LOCAL CONST Robtarget Tr_meulage_motif_1_166 := [[-76.86,48.46900390625,71.8286484375],[0.376363228761976,-0.369466106511504,0.595187364718739,-0.60629820802494],[0,0,0,0],[8.999999E+09,8.999999E+09,8.999999E+09,8.999999E+09,8.999999E+09,8.999999E+09]];
    LOCAL CONST Robtarget Tr_meulage_motif_1_167 := [[-77.2956796875,47.56890234375,71.8286484375],[0.376363228761976,-0.369466106511504,0.595187364718739,-0.60629820802494],[0,0,0,0],[8.999999E+09,8.999999E+09,8.999999E+09,8.999999E+09,8.999999E+09,8.999999E+09]];
    LOCAL CONST Robtarget Tr_meulage_motif_1_168 := [[-77.7313671875,46.6688046875,71.82865625],[0.376363228761976,-0.369466106511504,0.595187364718739,-0.60629820802494],[0,0,0,0],[8.999999E+09,8.999999E+09,8.999999E+09,8.999999E+09,8.999999E+09,8.999999E+09]];
    LOCAL CONST Robtarget Tr_meulage_motif_1_169 := [[-78.167046875,45.768703125,71.82865625],[0.376363228761976,-0.369466106511504,0.595187364718739,-0.60629820802494],[0,0,0,0],[8.999999E+09,8.999999E+09,8.999999E+09,8.999999E+09,8.999999E+09,8.999999E+09]];
    LOCAL CONST Robtarget Tr_meulage_motif_1_170 := [[-78.602734375,44.86860546875,71.82865625],[0.376363228761976,-0.369466106511504,0.595187364718739,-0.60629820802494],[0,0,0,0],[8.999999E+09,8.999999E+09,8.999999E+09,8.999999E+09,8.999999E+09,8.999999E+09]];
    LOCAL CONST Robtarget Tr_meulage_motif_1_171 := [[-79.038421875,43.96850390625,71.8286640625],[0.376363228761976,-0.369466106511504,0.595187364718739,-0.60629820802494],[0,0,0,0],[8.999999E+09,8.999999E+09,8.999999E+09,8.999999E+09,8.999999E+09,8.999999E+09]];
    LOCAL CONST Robtarget Tr_meulage_motif_1_172 := [[-79.4741015625,43.06840625,71.8286640625],[0.376363228761976,-0.369466106511504,0.595187364718739,-0.60629820802494],[0,0,0,0],[8.999999E+09,8.999999E+09,8.999999E+09,8.999999E+09,8.999999E+09,8.999999E+09]];
    LOCAL CONST Robtarget Tr_meulage_motif_1_173 := [[-79.9097890625,42.1683046875,71.828671875],[0.376363228761976,-0.369466106511504,0.595187364718739,-0.60629820802494],[0,0,0,0],[8.999999E+09,8.999999E+09,8.999999E+09,8.999999E+09,8.999999E+09,8.999999E+09]];
    LOCAL CONST Robtarget Tr_meulage_motif_1_174 := [[-80.34546875,41.26820703125,71.828671875],[0.376363228761976,-0.369466106511504,0.595187364718739,-0.60629820802494],[0,0,0,0],[8.999999E+09,8.999999E+09,8.999999E+09,8.999999E+09,8.999999E+09,8.999999E+09]];
    LOCAL CONST Robtarget Tr_meulage_motif_1_175 := [[-80.78115625,40.36810546875,71.8286796875],[0.376363228761976,-0.369466106511504,0.595187364718739,-0.60629820802494],[0,0,0,0],[8.999999E+09,8.999999E+09,8.999999E+09,8.999999E+09,8.999999E+09,8.999999E+09]];
    LOCAL CONST Robtarget Tr_meulage_motif_1_176 := [[-81.2168359375,39.4680078125,71.8286796875],[0.376363228761976,-0.369466106511504,0.595187364718739,-0.60629820802494],[0,0,0,0],[8.999999E+09,8.999999E+09,8.999999E+09,8.999999E+09,8.999999E+09,8.999999E+09]];
    LOCAL CONST Robtarget Tr_meulage_motif_1_177 := [[-81.6525234375,38.56790625,71.8286796875],[0.376363228761976,-0.369466106511504,0.595187364718739,-0.60629820802494],[0,0,0,0],[8.999999E+09,8.999999E+09,8.999999E+09,8.999999E+09,8.999999E+09,8.999999E+09]];
    LOCAL CONST Robtarget Tr_meulage_motif_1_178 := [[-82.0882109375,37.66780859375,71.8286875],[0.376363228761976,-0.369466106511504,0.595187364718739,-0.60629820802494],[0,0,0,0],[8.999999E+09,8.999999E+09,8.999999E+09,8.999999E+09,8.999999E+09,8.999999E+09]];
    LOCAL CONST Robtarget Tr_meulage_motif_1_179 := [[-82.523890625,36.76770703125,71.8286875],[0.376363228761976,-0.369466106511504,0.595187364718739,-0.60629820802494],[0,0,0,0],[8.999999E+09,8.999999E+09,8.999999E+09,8.999999E+09,8.999999E+09,8.999999E+09]];
    LOCAL CONST Robtarget Tr_meulage_motif_1_180 := [[-82.959578125,35.867609375,71.8286953125],[0.376363228761976,-0.369466106511504,0.595187364718739,-0.60629820802494],[0,0,0,0],[8.999999E+09,8.999999E+09,8.999999E+09,8.999999E+09,8.999999E+09,8.999999E+09]];
    LOCAL CONST Robtarget Tr_meulage_motif_1_181 := [[-83.3952578125,34.9675078125,71.8286953125],[0.376363228761976,-0.369466106511504,0.595187364718739,-0.60629820802494],[0,0,0,0],[8.999999E+09,8.999999E+09,8.999999E+09,8.999999E+09,8.999999E+09,8.999999E+09]];
    LOCAL CONST Robtarget Tr_meulage_motif_1_182 := [[-83.8309453125,34.06741015625,71.828703125],[0.376363228761976,-0.369466106511504,0.595187364718739,-0.60629820802494],[0,0,0,0],[8.999999E+09,8.999999E+09,8.999999E+09,8.999999E+09,8.999999E+09,8.999999E+09]];
    LOCAL CONST Robtarget Tr_meulage_motif_1_183 := [[-84.2666328125,33.16730859375,71.828703125],[0.376363228761976,-0.369466106511504,0.595187364718739,-0.60629820802494],[0,0,0,0],[8.999999E+09,8.999999E+09,8.999999E+09,8.999999E+09,8.999999E+09,8.999999E+09]];
    LOCAL CONST Robtarget Tr_meulage_motif_1_184 := [[-84.7023125,32.2672109375,71.828703125],[0.376363228761976,-0.369466106511504,0.595187364718739,-0.60629820802494],[0,0,0,0],[8.999999E+09,8.999999E+09,8.999999E+09,8.999999E+09,8.999999E+09,8.999999E+09]];
    LOCAL CONST Robtarget Tr_meulage_motif_1_185 := [[-85.138,31.367111328125,71.8287109375],[0.376363228761976,-0.369466106511504,0.595187364718739,-0.60629820802494],[0,0,0,0],[8.999999E+09,8.999999E+09,8.999999E+09,8.999999E+09,8.999999E+09,8.999999E+09]];
    LOCAL CONST Robtarget Tr_meulage_motif_1_186 := [[-85.570015625,30.473498046875,71.7181171875],[0.376363228761976,-0.369466106511504,0.595187364718739,-0.60629820802494],[0,0,0,0],[8.999999E+09,8.999999E+09,8.999999E+09,8.999999E+09,8.999999E+09,8.999999E+09]];
    LOCAL CONST Robtarget Tr_meulage_motif_1_187 := [[-85.981578125,29.62116015625,71.5069375],[0.376363228761976,-0.369466106511504,0.595187364718739,-0.60629820802494],[0,0,0,0],[8.999999E+09,8.999999E+09,8.999999E+09,8.999999E+09,8.999999E+09,8.999999E+09]];
    LOCAL CONST Robtarget Tr_meulage_motif_1_188 := [[-86.352046875,28.853119140625,71.2351015625],[0.376363228761976,-0.369466106511504,0.595187364718739,-0.60629820802494],[0,0,0,0],[8.999999E+09,8.999999E+09,8.999999E+09,8.999999E+09,8.999999E+09,8.999999E+09]];
    LOCAL CONST Robtarget Tr_meulage_motif_1_189 := [[-86.67771875,28.1775859375,70.9591640625],[0.376363228761976,-0.369466106511504,0.595187364718739,-0.60629820802494],[0,0,0,0],[8.999999E+09,8.999999E+09,8.999999E+09,8.999999E+09,8.999999E+09,8.999999E+09]];
    LOCAL CONST Robtarget Tr_meulage_motif_1_190 := [[-87.1550546875,27.1853671875,70.3430546875],[0.376363228761976,-0.369466106511504,0.595187364718739,-0.60629820802494],[0,0,0,0],[8.999999E+09,8.999999E+09,8.999999E+09,8.999999E+09,8.999999E+09,8.999999E+09]];
    LOCAL CONST Robtarget Tr_meulage_motif_1_191 := [[-87.597875,26.262193359375,69.49540625],[0.376363228761976,-0.369466106511504,0.595187364718739,-0.60629820802494],[0,0,0,0],[8.999999E+09,8.999999E+09,8.999999E+09,8.999999E+09,8.999999E+09,8.999999E+09]];
    LOCAL CONST Robtarget Tr_meulage_motif_1_192 := [[-87.963234375,25.497302734375,68.471546875],[0.376363228761976,-0.369466106511504,0.595187364718739,-0.60629820802494],[0,0,0,0],[8.999999E+09,8.999999E+09,8.999999E+09,8.999999E+09,8.999999E+09,8.999999E+09]];
    LOCAL CONST Robtarget Tr_meulage_motif_1_193 := [[-88.1716171875,25.055826171875,67.3553671875],[0.376363228761976,-0.369466106511504,0.595187364718739,-0.60629820802494],[0,0,0,0],[8.999999E+09,8.999999E+09,8.999999E+09,8.999999E+09,8.999999E+09,8.999999E+09]];
    LOCAL CONST Robtarget Tr_meulage_motif_1_194 := [[-88.1807265625,25.030166015625,66.65940625],[0.376363228761976,-0.369466106511504,0.595187364718739,-0.60629820802494],[0,0,0,0],[8.999999E+09,8.999999E+09,8.999999E+09,8.999999E+09,8.999999E+09,8.999999E+09]];
    LOCAL CONST Robtarget Tr_meulage_motif_1_195 := [[-88.178171875,25.0289296875,65.9981640625],[0.376363228761976,-0.369466106511504,0.595187364718739,-0.60629820802494],[0,0,0,0],[8.999999E+09,8.999999E+09,8.999999E+09,8.999999E+09,8.999999E+09,8.999999E+09]];
    LOCAL CONST Robtarget Tr_meulage_motif_1_196 := [[-88.15171875,25.0770859375,65.33707421875],[0.376363228761976,-0.369466106511504,0.595187364718739,-0.60629820802494],[0,0,0,0],[8.999999E+09,8.999999E+09,8.999999E+09,8.999999E+09,8.999999E+09,8.999999E+09]];
    LOCAL CONST Robtarget Tr_meulage_motif_1_197 := [[-87.93040625,25.52347265625,64.23533203125],[0.376363228761976,-0.369466106511504,0.595187364718739,-0.60629820802494],[0,0,0,0],[8.999999E+09,8.999999E+09,8.999999E+09,8.999999E+09,8.999999E+09,8.999999E+09]];
    LOCAL CONST Robtarget Tr_meulage_motif_1_198 := [[-87.5533046875,26.292638671875,63.22871484375],[0.376363228761976,-0.369466106511504,0.595187364718739,-0.60629820802494],[0,0,0,0],[8.999999E+09,8.999999E+09,8.999999E+09,8.999999E+09,8.999999E+09,8.999999E+09]];
    LOCAL CONST Robtarget Tr_meulage_motif_1_199 := [[-87.1042265625,27.212255859375,62.39984375],[0.376363228761976,-0.369466106511504,0.595187364718739,-0.60629820802494],[0,0,0,0],[8.999999E+09,8.999999E+09,8.999999E+09,8.999999E+09,8.999999E+09,8.999999E+09]];
    LOCAL CONST Robtarget Tr_meulage_motif_1_200 := [[-86.80334375,27.82996875,62.00409375],[0.376363228761976,-0.369466106511504,0.595187364718739,-0.60629820802494],[0,0,0,0],[8.999999E+09,8.999999E+09,8.999999E+09,8.999999E+09,8.999999E+09,8.999999E+09]];
    LOCAL CONST Robtarget Tr_meulage_motif_1_201 := [[-86.296875,28.871513671875,61.5165625],[0.376363228761976,-0.369466106511504,0.595187364718739,-0.60629820802494],[0,0,0,0],[8.999999E+09,8.999999E+09,8.999999E+09,8.999999E+09,8.999999E+09,8.999999E+09]];
    LOCAL CONST Robtarget Tr_meulage_motif_1_202 := [[-85.9276875,29.631630859375,61.25246875],[0.376363228761976,-0.369466106511504,0.595187364718739,-0.60629820802494],[0,0,0,0],[8.999999E+09,8.999999E+09,8.999999E+09,8.999999E+09,8.999999E+09,8.999999E+09]];
    LOCAL CONST Robtarget Tr_meulage_motif_1_203 := [[-85.52084375,30.470142578125,61.048],[0.376363228761976,-0.369466106511504,0.595187364718739,-0.60629820802494],[0,0,0,0],[8.999999E+09,8.999999E+09,8.999999E+09,8.999999E+09,8.999999E+09,8.999999E+09]];
    LOCAL CONST Robtarget Tr_meulage_motif_1_204 := [[-85.0927734375,31.353443359375,60.93940234375],[0.376363228761976,-0.369466106511504,0.595187364718739,-0.60629820802494],[0,0,0,0],[8.999999E+09,8.999999E+09,8.999999E+09,8.999999E+09,8.999999E+09,8.999999E+09]];
    LOCAL CONST Robtarget Tr_meulage_motif_1_205 := [[-84.65990625,32.246640625,60.82880859375],[0.376363228761976,-0.369466106511504,0.595187364718739,-0.60629820802494],[0,0,0,0],[8.999999E+09,8.999999E+09,8.999999E+09,8.999999E+09,8.999999E+09,8.999999E+09]];
    LOCAL CONST Robtarget Tr_meulage_motif_1_206 := [[-84.22421875,33.1467421875,60.8288046875],[0.376363228761976,-0.369466106511504,0.595187364718739,-0.60629820802494],[0,0,0,0],[8.999999E+09,8.999999E+09,8.999999E+09,8.999999E+09,8.999999E+09,8.999999E+09]];
    LOCAL CONST Robtarget Tr_meulage_motif_1_207 := [[-83.78853125,34.04683984375,60.82880078125],[0.376363228761976,-0.369466106511504,0.595187364718739,-0.60629820802494],[0,0,0,0],[8.999999E+09,8.999999E+09,8.999999E+09,8.999999E+09,8.999999E+09,8.999999E+09]];
    LOCAL CONST Robtarget Tr_meulage_motif_1_208 := [[-83.3528515625,34.94694140625,60.828796875],[0.376363228761976,-0.369466106511504,0.595187364718739,-0.60629820802494],[0,0,0,0],[8.999999E+09,8.999999E+09,8.999999E+09,8.999999E+09,8.999999E+09,8.999999E+09]];
    LOCAL CONST Robtarget Tr_meulage_motif_1_209 := [[-82.9171640625,35.8470390625,60.82879296875],[0.376363228761976,-0.369466106511504,0.595187364718739,-0.60629820802494],[0,0,0,0],[8.999999E+09,8.999999E+09,8.999999E+09,8.999999E+09,8.999999E+09,8.999999E+09]];
    LOCAL CONST Robtarget Tr_meulage_motif_1_210 := [[-82.481484375,36.747140625,60.8287890625],[0.376363228761976,-0.369466106511504,0.595187364718739,-0.60629820802494],[0,0,0,0],[8.999999E+09,8.999999E+09,8.999999E+09,8.999999E+09,8.999999E+09,8.999999E+09]];
    LOCAL CONST Robtarget Tr_meulage_motif_1_211 := [[-82.045796875,37.64723828125,60.82878515625],[0.376363228761976,-0.369466106511504,0.595187364718739,-0.60629820802494],[0,0,0,0],[8.999999E+09,8.999999E+09,8.999999E+09,8.999999E+09,8.999999E+09,8.999999E+09]];
    LOCAL CONST Robtarget Tr_meulage_motif_1_212 := [[-81.610109375,38.5473359375,60.82878515625],[0.376363228761976,-0.369466106511504,0.595187364718739,-0.60629820802494],[0,0,0,0],[8.999999E+09,8.999999E+09,8.999999E+09,8.999999E+09,8.999999E+09,8.999999E+09]];
    LOCAL CONST Robtarget Tr_meulage_motif_1_213 := [[-81.1744296875,39.4474375,60.82878125],[0.376363228761976,-0.369466106511504,0.595187364718739,-0.60629820802494],[0,0,0,0],[8.999999E+09,8.999999E+09,8.999999E+09,8.999999E+09,8.999999E+09,8.999999E+09]];
    LOCAL CONST Robtarget Tr_meulage_motif_1_214 := [[-80.7387421875,40.34753515625,60.82877734375],[0.376363228761976,-0.369466106511504,0.595187364718739,-0.60629820802494],[0,0,0,0],[8.999999E+09,8.999999E+09,8.999999E+09,8.999999E+09,8.999999E+09,8.999999E+09]];
    LOCAL CONST Robtarget Tr_meulage_motif_1_215 := [[-80.3030625,41.24763671875,60.8287734375],[0.376363228761976,-0.369466106511504,0.595187364718739,-0.60629820802494],[0,0,0,0],[8.999999E+09,8.999999E+09,8.999999E+09,8.999999E+09,8.999999E+09,8.999999E+09]];
    LOCAL CONST Robtarget Tr_meulage_motif_1_216 := [[-79.867375,42.147734375,60.82876953125],[0.376363228761976,-0.369466106511504,0.595187364718739,-0.60629820802494],[0,0,0,0],[8.999999E+09,8.999999E+09,8.999999E+09,8.999999E+09,8.999999E+09,8.999999E+09]];
    LOCAL CONST Robtarget Tr_meulage_motif_1_217 := [[-79.4316953125,43.0478359375,60.828765625],[0.376363228761976,-0.369466106511504,0.595187364718739,-0.60629820802494],[0,0,0,0],[8.999999E+09,8.999999E+09,8.999999E+09,8.999999E+09,8.999999E+09,8.999999E+09]];
    LOCAL CONST Robtarget Tr_meulage_motif_1_218 := [[-78.9960078125,43.94793359375,60.82876171875],[0.376363228761976,-0.369466106511504,0.595187364718739,-0.60629820802494],[0,0,0,0],[8.999999E+09,8.999999E+09,8.999999E+09,8.999999E+09,8.999999E+09,8.999999E+09]];
    LOCAL CONST Robtarget Tr_meulage_motif_1_219 := [[-78.5603203125,44.84803515625,60.82876171875],[0.376363228761976,-0.369466106511504,0.595187364718739,-0.60629820802494],[0,0,0,0],[8.999999E+09,8.999999E+09,8.999999E+09,8.999999E+09,8.999999E+09,8.999999E+09]];
    LOCAL CONST Robtarget Tr_meulage_motif_1_220 := [[-78.124640625,45.7481328125,60.8287578125],[0.376363228761976,-0.369466106511504,0.595187364718739,-0.60629820802494],[0,0,0,0],[8.999999E+09,8.999999E+09,8.999999E+09,8.999999E+09,8.999999E+09,8.999999E+09]];
    LOCAL CONST Robtarget Tr_meulage_motif_1_221 := [[-77.688953125,46.648234375,60.82875390625],[0.376363228761976,-0.369466106511504,0.595187364718739,-0.60629820802494],[0,0,0,0],[8.999999E+09,8.999999E+09,8.999999E+09,8.999999E+09,8.999999E+09,8.999999E+09]];
    LOCAL CONST Robtarget Tr_meulage_motif_1_222 := [[-77.2532734375,47.54833203125,60.82875],[0.376363228761976,-0.369466106511504,0.595187364718739,-0.60629820802494],[0,0,0,0],[8.999999E+09,8.999999E+09,8.999999E+09,8.999999E+09,8.999999E+09,8.999999E+09]];
    LOCAL CONST Robtarget Tr_meulage_motif_1_223 := [[-76.8175859375,48.44843359375,60.82874609375],[0.376363228761976,-0.369466106511504,0.595187364718739,-0.60629820802494],[0,0,0,0],[8.999999E+09,8.999999E+09,8.999999E+09,8.999999E+09,8.999999E+09,8.999999E+09]];
    LOCAL CONST Robtarget Tr_meulage_motif_1_224 := [[-76.3818984375,49.34853125,60.8287421875],[0.376363228761976,-0.369466106511504,0.595187364718739,-0.60629820802494],[0,0,0,0],[8.999999E+09,8.999999E+09,8.999999E+09,8.999999E+09,8.999999E+09,8.999999E+09]];
    LOCAL CONST Robtarget Tr_meulage_motif_1_225 := [[-75.94621875,50.2486328125,60.82873828125],[0.376363228761976,-0.369466106511504,0.595187364718739,-0.60629820802494],[0,0,0,0],[8.999999E+09,8.999999E+09,8.999999E+09,8.999999E+09,8.999999E+09,8.999999E+09]];
    LOCAL CONST Robtarget Tr_meulage_motif_1_226 := [[-75.51053125,51.14873046875,60.82873828125],[0.376363228761976,-0.369466106511504,0.595187364718739,-0.60629820802494],[0,0,0,0],[8.999999E+09,8.999999E+09,8.999999E+09,8.999999E+09,8.999999E+09,8.999999E+09]];
    LOCAL CONST Robtarget Tr_meulage_motif_1_227 := [[-75.0748515625,52.04883203125,60.828734375],[0.376363228761976,-0.369466106511504,0.595187364718739,-0.60629820802494],[0,0,0,0],[8.999999E+09,8.999999E+09,8.999999E+09,8.999999E+09,8.999999E+09,8.999999E+09]];
    LOCAL CONST Robtarget Tr_meulage_motif_1_228 := [[-74.6391640625,52.9489296875,60.82873046875],[0.376363228761976,-0.369466106511504,0.595187364718739,-0.60629820802494],[0,0,0,0],[8.999999E+09,8.999999E+09,8.999999E+09,8.999999E+09,8.999999E+09,8.999999E+09]];
    LOCAL CONST Robtarget Tr_meulage_motif_1_229 := [[-74.203484375,53.84903125,60.8287265625],[0.376363228761976,-0.369466106511504,0.595187364718739,-0.60629820802494],[0,0,0,0],[8.999999E+09,8.999999E+09,8.999999E+09,8.999999E+09,8.999999E+09,8.999999E+09]];
    LOCAL CONST Robtarget Tr_meulage_motif_1_230 := [[-73.767796875,54.74912890625,60.82872265625],[0.376363228761976,-0.369466106511504,0.595187364718739,-0.60629820802494],[0,0,0,0],[8.999999E+09,8.999999E+09,8.999999E+09,8.999999E+09,8.999999E+09,8.999999E+09]];
    LOCAL CONST Robtarget Tr_meulage_motif_1_231 := [[-73.332109375,55.64923046875,60.82871875],[0.376363228761976,-0.369466106511504,0.595187364718739,-0.60629820802494],[0,0,0,0],[8.999999E+09,8.999999E+09,8.999999E+09,8.999999E+09,8.999999E+09,8.999999E+09]];
    LOCAL CONST Robtarget Tr_meulage_motif_1_232 := [[-72.8964296875,56.549328125,60.82871484375],[0.376363228761976,-0.369466106511504,0.595187364718739,-0.60629820802494],[0,0,0,0],[8.999999E+09,8.999999E+09,8.999999E+09,8.999999E+09,8.999999E+09,8.999999E+09]];
    LOCAL CONST Robtarget Tr_meulage_motif_1_233 := [[-72.4607421875,57.4494296875,60.82871484375],[0.376363228761976,-0.369466106511504,0.595187364718739,-0.60629820802494],[0,0,0,0],[8.999999E+09,8.999999E+09,8.999999E+09,8.999999E+09,8.999999E+09,8.999999E+09]];
    LOCAL CONST Robtarget Tr_meulage_motif_1_234 := [[-72.0250625,58.34952734375,60.8287109375],[0.376363228761976,-0.369466106511504,0.595187364718739,-0.60629820802494],[0,0,0,0],[8.999999E+09,8.999999E+09,8.999999E+09,8.999999E+09,8.999999E+09,8.999999E+09]];
    LOCAL CONST Robtarget Tr_meulage_motif_1_235 := [[-71.589375,59.24962890625,60.82870703125],[0.376363228761976,-0.369466106511504,0.595187364718739,-0.60629820802494],[0,0,0,0],[8.999999E+09,8.999999E+09,8.999999E+09,8.999999E+09,8.999999E+09,8.999999E+09]];
    LOCAL CONST Robtarget Tr_meulage_motif_1_236 := [[-71.1536875,60.1497265625,60.828703125],[0.376363228761976,-0.369466106511504,0.595187364718739,-0.60629820802494],[0,0,0,0],[8.999999E+09,8.999999E+09,8.999999E+09,8.999999E+09,8.999999E+09,8.999999E+09]];
    LOCAL CONST Robtarget Tr_meulage_motif_1_237 := [[-70.7180078125,61.049828125,60.82869921875],[0.376363228761976,-0.369466106511504,0.595187364718739,-0.60629820802494],[0,0,0,0],[8.999999E+09,8.999999E+09,8.999999E+09,8.999999E+09,8.999999E+09,8.999999E+09]];
    LOCAL CONST Robtarget Tr_meulage_motif_1_238 := [[-70.2823203125,61.94992578125,60.8286953125],[0.376363228761976,-0.369466106511504,0.595187364718739,-0.60629820802494],[0,0,0,0],[8.999999E+09,8.999999E+09,8.999999E+09,8.999999E+09,8.999999E+09,8.999999E+09]];
    LOCAL CONST Robtarget Tr_meulage_motif_1_239 := [[-69.846640625,62.85002734375,60.82869140625],[0.376363228761976,-0.369466106511504,0.595187364718739,-0.60629820802494],[0,0,0,0],[8.999999E+09,8.999999E+09,8.999999E+09,8.999999E+09,8.999999E+09,8.999999E+09]];
    LOCAL CONST Robtarget Tr_meulage_motif_1_240 := [[-69.410953125,63.750125,60.82869140625],[0.376363228761976,-0.369466106511504,0.595187364718739,-0.60629820802494],[0,0,0,0],[8.999999E+09,8.999999E+09,8.999999E+09,8.999999E+09,8.999999E+09,8.999999E+09]];
    LOCAL CONST Robtarget Tr_meulage_motif_1_241 := [[-68.9752734375,64.6502265625,60.8286875],[0.376363228761976,-0.369466106511504,0.595187364718739,-0.60629820802494],[0,0,0,0],[8.999999E+09,8.999999E+09,8.999999E+09,8.999999E+09,8.999999E+09,8.999999E+09]];
    LOCAL CONST Robtarget Tr_meulage_motif_1_242 := [[-68.5395859375,65.550328125,60.82868359375],[0.376363228761976,-0.369466106511504,0.595187364718739,-0.60629820802494],[0,0,0,0],[8.999999E+09,8.999999E+09,8.999999E+09,8.999999E+09,8.999999E+09,8.999999E+09]];
    LOCAL CONST Robtarget Tr_meulage_motif_1_243 := [[-68.1038984375,66.450421875,60.8286796875],[0.376363228761976,-0.369466106511504,0.595187364718739,-0.60629820802494],[0,0,0,0],[8.999999E+09,8.999999E+09,8.999999E+09,8.999999E+09,8.999999E+09,8.999999E+09]];
    LOCAL CONST Robtarget Tr_meulage_motif_1_244 := [[-67.66821875,67.3505234375,60.82867578125],[0.376363228761976,-0.369466106511504,0.595187364718739,-0.60629820802494],[0,0,0,0],[8.999999E+09,8.999999E+09,8.999999E+09,8.999999E+09,8.999999E+09,8.999999E+09]];
    LOCAL CONST Robtarget Tr_meulage_motif_1_245 := [[-67.23253125,68.250625,60.828671875],[0.376363228761976,-0.369466106511504,0.595187364718739,-0.60629820802494],[0,0,0,0],[8.999999E+09,8.999999E+09,8.999999E+09,8.999999E+09,8.999999E+09,8.999999E+09]];
    LOCAL CONST Robtarget Tr_meulage_motif_1_246 := [[-66.7968515625,69.1507265625,60.82866796875],[0.376363228761976,-0.369466106511504,0.595187364718739,-0.60629820802494],[0,0,0,0],[8.999999E+09,8.999999E+09,8.999999E+09,8.999999E+09,8.999999E+09,8.999999E+09]];
    LOCAL CONST Robtarget Tr_meulage_motif_1_247 := [[-66.3611640625,70.0508203125,60.82866796875],[0.376363228761976,-0.369466106511504,0.595187364718739,-0.60629820802494],[0,0,0,0],[8.999999E+09,8.999999E+09,8.999999E+09,8.999999E+09,8.999999E+09,8.999999E+09]];
    LOCAL CONST Robtarget Tr_meulage_motif_1_248 := [[-65.9254765625,70.950921875,60.8286640625],[0.376363228761976,-0.369466106511504,0.595187364718739,-0.60629820802494],[0,0,0,0],[8.999999E+09,8.999999E+09,8.999999E+09,8.999999E+09,8.999999E+09,8.999999E+09]];
    LOCAL CONST Robtarget Tr_meulage_motif_1_249 := [[-65.489796875,71.8510234375,60.82866015625],[0.376363228761976,-0.369466106511504,0.595187364718739,-0.60629820802494],[0,0,0,0],[8.999999E+09,8.999999E+09,8.999999E+09,8.999999E+09,8.999999E+09,8.999999E+09]];
    LOCAL CONST Robtarget Tr_meulage_motif_1_250 := [[-65.05411328125,72.751125,60.82865625],[0.376363228761976,-0.369466106511504,0.595187364718739,-0.60629820802494],[0,0,0,0],[8.999999E+09,8.999999E+09,8.999999E+09,8.999999E+09,8.999999E+09,8.999999E+09]];
    LOCAL CONST Robtarget Tr_meulage_motif_1_251 := [[-64.61842578125,73.65121875,60.82865234375],[0.376363228761976,-0.369466106511504,0.595187364718739,-0.60629820802494],[0,0,0,0],[8.999999E+09,8.999999E+09,8.999999E+09,8.999999E+09,8.999999E+09,8.999999E+09]];
    LOCAL CONST Robtarget Tr_meulage_motif_1_252 := [[-64.18555859375,74.544421875,60.71805859375],[0.376363228761976,-0.369466106511504,0.595187364718739,-0.60629820802494],[0,0,0,0],[8.999999E+09,8.999999E+09,8.999999E+09,8.999999E+09,8.999999E+09,8.999999E+09]];
    LOCAL CONST Robtarget Tr_meulage_motif_1_253 := [[-63.7723671875,75.39596875,60.5068671875],[0.376363228761976,-0.369466106511504,0.595187364718739,-0.60629820802494],[0,0,0,0],[8.999999E+09,8.999999E+09,8.999999E+09,8.999999E+09,8.999999E+09,8.999999E+09]];
    LOCAL CONST Robtarget Tr_meulage_motif_1_254 := [[-63.3998046875,76.1629921875,60.2350234375],[0.376363228761976,-0.369466106511504,0.595187364718739,-0.60629820802494],[0,0,0,0],[8.999999E+09,8.999999E+09,8.999999E+09,8.999999E+09,8.999999E+09,8.999999E+09]];
    LOCAL CONST Robtarget Tr_meulage_motif_1_255 := [[-63.088640625,76.80284375,59.9308828125],[0.376363228761976,-0.369466106511504,0.595187364718739,-0.60629820802494],[0,0,0,0],[8.999999E+09,8.999999E+09,8.999999E+09,8.999999E+09,8.999999E+09,8.999999E+09]];
    LOCAL CONST Robtarget Tr_meulage_motif_1_256 := [[-62.63538671875,77.7327265625,59.26835546875],[0.376363228761976,-0.369466106511504,0.595187364718739,-0.60629820802494],[0,0,0,0],[8.999999E+09,8.999999E+09,8.999999E+09,8.999999E+09,8.999999E+09,8.999999E+09]];
    LOCAL CONST Robtarget Tr_meulage_motif_1_257 := [[-62.23894921875,78.542875,58.36640625],[0.376363228761976,-0.369466106511504,0.595187364718739,-0.60629820802494],[0,0,0,0],[8.999999E+09,8.999999E+09,8.999999E+09,8.999999E+09,8.999999E+09,8.999999E+09]];
    LOCAL CONST Robtarget Tr_meulage_motif_1_258 := [[-62.0018359375,79.0224453125,57.3203984375],[0.376363228761976,-0.369466106511504,0.595187364718739,-0.60629820802494],[0,0,0,0],[8.999999E+09,8.999999E+09,8.999999E+09,8.999999E+09,8.999999E+09,8.999999E+09]];
    LOCAL CONST Robtarget Tr_meulage_motif_1_259 := [[-61.91866015625,79.18746875,56.627171875],[0.376363228761976,-0.369466106511504,0.595187364718739,-0.60629820802494],[0,0,0,0],[8.999999E+09,8.999999E+09,8.999999E+09,8.999999E+09,8.999999E+09,8.999999E+09]];
    LOCAL CONST Robtarget Tr_meulage_motif_1_260 := [[-61.887875,79.2435,55.8571796875],[0.376363228761976,-0.369466106511504,0.595187364718739,-0.60629820802494],[0,0,0,0],[8.999999E+09,8.999999E+09,8.999999E+09,8.999999E+09,8.999999E+09,8.999999E+09]];
    LOCAL CONST Robtarget Tr_meulage_motif_1_261 := [[-61.9140703125,79.1818046875,55.08732421875],[0.376363228761976,-0.369466106511504,0.595187364718739,-0.60629820802494],[0,0,0,0],[8.999999E+09,8.999999E+09,8.999999E+09,8.999999E+09,8.999999E+09,8.999999E+09]];
    LOCAL CONST Robtarget Tr_meulage_motif_1_262 := [[-62.09260546875,78.8020625,53.9790859375],[0.376363228761976,-0.369466106511504,0.595187364718739,-0.60629820802494],[0,0,0,0],[8.999999E+09,8.999999E+09,8.999999E+09,8.999999E+09,8.999999E+09,8.999999E+09]];
    LOCAL CONST Robtarget Tr_meulage_motif_1_263 := [[-62.270859375,78.4280390625,53.39340625],[0.376363228761976,-0.369466106511504,0.595187364718739,-0.60629820802494],[0,0,0,0],[8.999999E+09,8.999999E+09,8.999999E+09,8.999999E+09,8.999999E+09,8.999999E+09]];
    LOCAL CONST Robtarget Tr_meulage_motif_1_264 := [[-62.6539453125,77.6278828125,52.50626171875],[0.376363228761976,-0.369466106511504,0.595187364718739,-0.60629820802494],[0,0,0,0],[8.999999E+09,8.999999E+09,8.999999E+09,8.999999E+09,8.999999E+09,8.999999E+09]];
    LOCAL CONST Robtarget Tr_meulage_motif_1_265 := [[-62.9075234375,77.0999296875,52.091984375],[0.376363228761976,-0.369466106511504,0.595187364718739,-0.60629820802494],[0,0,0,0],[8.999999E+09,8.999999E+09,8.999999E+09,8.999999E+09,8.999999E+09,8.999999E+09]];
    LOCAL CONST Robtarget Tr_meulage_motif_1_266 := [[-63.3924765625,76.0926875,51.54787109375],[0.376363228761976,-0.369466106511504,0.595187364718739,-0.60629820802494],[0,0,0,0],[8.999999E+09,8.999999E+09,8.999999E+09,8.999999E+09,8.999999E+09,8.999999E+09]];
    LOCAL CONST Robtarget Tr_meulage_motif_1_267 := [[-63.75103515625,75.349015625,51.252375],[0.376363228761976,-0.369466106511504,0.595187364718739,-0.60629820802494],[0,0,0,0],[8.999999E+09,8.999999E+09,8.999999E+09,8.999999E+09,8.999999E+09,8.999999E+09]];
    LOCAL CONST Robtarget Tr_meulage_motif_1_268 := [[-64.1563046875,74.5097421875,51.04789453125],[0.376363228761976,-0.369466106511504,0.595187364718739,-0.60629820802494],[0,0,0,0],[8.999999E+09,8.999999E+09,8.999999E+09,8.999999E+09,8.999999E+09,8.999999E+09]];
    LOCAL CONST Robtarget Tr_meulage_motif_1_269 := [[-64.5835390625,73.62603125,50.9393515625],[0.376363228761976,-0.369466106511504,0.595187364718739,-0.60629820802494],[0,0,0,0],[8.999999E+09,8.999999E+09,8.999999E+09,8.999999E+09,8.999999E+09,8.999999E+09]];
    LOCAL CONST Robtarget Tr_meulage_motif_1_270 := [[-65.0155546875,72.732421875,50.82875],[0.376363228761976,-0.369466106511504,0.595187364718739,-0.60629820802494],[0,0,0,0],[8.999999E+09,8.999999E+09,8.999999E+09,8.999999E+09,8.999999E+09,8.999999E+09]];
    LOCAL CONST Robtarget Tr_meulage_motif_1_271 := [[-65.4512421875,71.8323203125,50.82875],[0.376363228761976,-0.369466106511504,0.595187364718739,-0.60629820802494],[0,0,0,0],[8.999999E+09,8.999999E+09,8.999999E+09,8.999999E+09,8.999999E+09,8.999999E+09]];
    LOCAL CONST Robtarget Tr_meulage_motif_1_272 := [[-65.886921875,70.9322265625,50.82875390625],[0.376363228761976,-0.369466106511504,0.595187364718739,-0.60629820802494],[0,0,0,0],[8.999999E+09,8.999999E+09,8.999999E+09,8.999999E+09,8.999999E+09,8.999999E+09]];
    LOCAL CONST Robtarget Tr_meulage_motif_1_273 := [[-66.322609375,70.032125,50.8287578125],[0.376363228761976,-0.369466106511504,0.595187364718739,-0.60629820802494],[0,0,0,0],[8.999999E+09,8.999999E+09,8.999999E+09,8.999999E+09,8.999999E+09,8.999999E+09]];
    LOCAL CONST Robtarget Tr_meulage_motif_1_274 := [[-66.758296875,69.1320234375,50.82876171875],[0.376363228761976,-0.369466106511504,0.595187364718739,-0.60629820802494],[0,0,0,0],[8.999999E+09,8.999999E+09,8.999999E+09,8.999999E+09,8.999999E+09,8.999999E+09]];
    LOCAL CONST Robtarget Tr_meulage_motif_1_275 := [[-67.1939765625,68.231921875,50.828765625],[0.376363228761976,-0.369466106511504,0.595187364718739,-0.60629820802494],[0,0,0,0],[8.999999E+09,8.999999E+09,8.999999E+09,8.999999E+09,8.999999E+09,8.999999E+09]];
    LOCAL CONST Robtarget Tr_meulage_motif_1_276 := [[-67.6296640625,67.331828125,50.82876953125],[0.376363228761976,-0.369466106511504,0.595187364718739,-0.60629820802494],[0,0,0,0],[8.999999E+09,8.999999E+09,8.999999E+09,8.999999E+09,8.999999E+09,8.999999E+09]];
    LOCAL CONST Robtarget Tr_meulage_motif_1_277 := [[-68.06534375,66.4317265625,50.8287734375],[0.376363228761976,-0.369466106511504,0.595187364718739,-0.60629820802494],[0,0,0,0],[8.999999E+09,8.999999E+09,8.999999E+09,8.999999E+09,8.999999E+09,8.999999E+09]];
    LOCAL CONST Robtarget Tr_meulage_motif_1_278 := [[-68.50103125,65.531625,50.8287734375],[0.376363228761976,-0.369466106511504,0.595187364718739,-0.60629820802494],[0,0,0,0],[8.999999E+09,8.999999E+09,8.999999E+09,8.999999E+09,8.999999E+09,8.999999E+09]];
    LOCAL CONST Robtarget Tr_meulage_motif_1_279 := [[-68.9367109375,64.63152734375,50.82877734375],[0.376363228761976,-0.369466106511504,0.595187364718739,-0.60629820802494],[0,0,0,0],[8.999999E+09,8.999999E+09,8.999999E+09,8.999999E+09,8.999999E+09,8.999999E+09]];
    LOCAL CONST Robtarget Tr_meulage_motif_1_280 := [[-69.3723984375,63.73142578125,50.82878125],[0.376363228761976,-0.369466106511504,0.595187364718739,-0.60629820802494],[0,0,0,0],[8.999999E+09,8.999999E+09,8.999999E+09,8.999999E+09,8.999999E+09,8.999999E+09]];
    LOCAL CONST Robtarget Tr_meulage_motif_1_281 := [[-69.8080859375,62.831328125,50.82878515625],[0.376363228761976,-0.369466106511504,0.595187364718739,-0.60629820802494],[0,0,0,0],[8.999999E+09,8.999999E+09,8.999999E+09,8.999999E+09,8.999999E+09,8.999999E+09]];
    LOCAL CONST Robtarget Tr_meulage_motif_1_282 := [[-70.243765625,61.9312265625,50.8287890625],[0.376363228761976,-0.369466106511504,0.595187364718739,-0.60629820802494],[0,0,0,0],[8.999999E+09,8.999999E+09,8.999999E+09,8.999999E+09,8.999999E+09,8.999999E+09]];
    LOCAL CONST Robtarget Tr_meulage_motif_1_283 := [[-70.679453125,61.03112890625,50.82879296875],[0.376363228761976,-0.369466106511504,0.595187364718739,-0.60629820802494],[0,0,0,0],[8.999999E+09,8.999999E+09,8.999999E+09,8.999999E+09,8.999999E+09,8.999999E+09]];
    LOCAL CONST Robtarget Tr_meulage_motif_1_284 := [[-71.1151328125,60.13102734375,50.828796875],[0.376363228761976,-0.369466106511504,0.595187364718739,-0.60629820802494],[0,0,0,0],[8.999999E+09,8.999999E+09,8.999999E+09,8.999999E+09,8.999999E+09,8.999999E+09]];
    LOCAL CONST Robtarget Tr_meulage_motif_1_285 := [[-71.5508203125,59.2309296875,50.828796875],[0.376363228761976,-0.369466106511504,0.595187364718739,-0.60629820802494],[0,0,0,0],[8.999999E+09,8.999999E+09,8.999999E+09,8.999999E+09,8.999999E+09,8.999999E+09]];
    LOCAL CONST Robtarget Tr_meulage_motif_1_286 := [[-71.9865078125,58.330828125,50.82880078125],[0.376363228761976,-0.369466106511504,0.595187364718739,-0.60629820802494],[0,0,0,0],[8.999999E+09,8.999999E+09,8.999999E+09,8.999999E+09,8.999999E+09,8.999999E+09]];
    LOCAL CONST Robtarget Tr_meulage_motif_1_287 := [[-72.4221875,57.43073046875,50.8288046875],[0.376363228761976,-0.369466106511504,0.595187364718739,-0.60629820802494],[0,0,0,0],[8.999999E+09,8.999999E+09,8.999999E+09,8.999999E+09,8.999999E+09,8.999999E+09]];
    LOCAL CONST Robtarget Tr_meulage_motif_1_288 := [[-72.857875,56.53062890625,50.82880859375],[0.376363228761976,-0.369466106511504,0.595187364718739,-0.60629820802494],[0,0,0,0],[8.999999E+09,8.999999E+09,8.999999E+09,8.999999E+09,8.999999E+09,8.999999E+09]];
    LOCAL CONST Robtarget Tr_meulage_motif_1_289 := [[-73.2935546875,55.63053125,50.8288125],[0.376363228761976,-0.369466106511504,0.595187364718739,-0.60629820802494],[0,0,0,0],[8.999999E+09,8.999999E+09,8.999999E+09,8.999999E+09,8.999999E+09,8.999999E+09]];
    LOCAL CONST Robtarget Tr_meulage_motif_1_290 := [[-73.7292421875,54.7304296875,50.82881640625],[0.376363228761976,-0.369466106511504,0.595187364718739,-0.60629820802494],[0,0,0,0],[8.999999E+09,8.999999E+09,8.999999E+09,8.999999E+09,8.999999E+09,8.999999E+09]];
    LOCAL CONST Robtarget Tr_meulage_motif_1_291 := [[-74.164921875,53.83033203125,50.8288203125],[0.376363228761976,-0.369466106511504,0.595187364718739,-0.60629820802494],[0,0,0,0],[8.999999E+09,8.999999E+09,8.999999E+09,8.999999E+09,8.999999E+09,8.999999E+09]];
    LOCAL CONST Robtarget Tr_meulage_motif_1_292 := [[-74.600609375,52.93023046875,50.8288203125],[0.376363228761976,-0.369466106511504,0.595187364718739,-0.60629820802494],[0,0,0,0],[8.999999E+09,8.999999E+09,8.999999E+09,8.999999E+09,8.999999E+09,8.999999E+09]];
    LOCAL CONST Robtarget Tr_meulage_motif_1_293 := [[-75.036296875,52.0301328125,50.82882421875],[0.376363228761976,-0.369466106511504,0.595187364718739,-0.60629820802494],[0,0,0,0],[8.999999E+09,8.999999E+09,8.999999E+09,8.999999E+09,8.999999E+09,8.999999E+09]];
    LOCAL CONST Robtarget Tr_meulage_motif_1_294 := [[-75.4719765625,51.13003125,50.828828125],[0.376363228761976,-0.369466106511504,0.595187364718739,-0.60629820802494],[0,0,0,0],[8.999999E+09,8.999999E+09,8.999999E+09,8.999999E+09,8.999999E+09,8.999999E+09]];
    LOCAL CONST Robtarget Tr_meulage_motif_1_295 := [[-75.9076640625,50.22993359375,50.82883203125],[0.376363228761976,-0.369466106511504,0.595187364718739,-0.60629820802494],[0,0,0,0],[8.999999E+09,8.999999E+09,8.999999E+09,8.999999E+09,8.999999E+09,8.999999E+09]];
    LOCAL CONST Robtarget Tr_meulage_motif_1_296 := [[-76.34334375,49.32983203125,50.8288359375],[0.376363228761976,-0.369466106511504,0.595187364718739,-0.60629820802494],[0,0,0,0],[8.999999E+09,8.999999E+09,8.999999E+09,8.999999E+09,8.999999E+09,8.999999E+09]];
    LOCAL CONST Robtarget Tr_meulage_motif_1_297 := [[-76.77903125,48.429734375,50.82883984375],[0.376363228761976,-0.369466106511504,0.595187364718739,-0.60629820802494],[0,0,0,0],[8.999999E+09,8.999999E+09,8.999999E+09,8.999999E+09,8.999999E+09,8.999999E+09]];
    LOCAL CONST Robtarget Tr_meulage_motif_1_298 := [[-77.21471875,47.5296328125,50.82884375],[0.376363228761976,-0.369466106511504,0.595187364718739,-0.60629820802494],[0,0,0,0],[8.999999E+09,8.999999E+09,8.999999E+09,8.999999E+09,8.999999E+09,8.999999E+09]];
    LOCAL CONST Robtarget Tr_meulage_motif_1_299 := [[-77.6503984375,46.62953515625,50.82884375],[0.376363228761976,-0.369466106511504,0.595187364718739,-0.60629820802494],[0,0,0,0],[8.999999E+09,8.999999E+09,8.999999E+09,8.999999E+09,8.999999E+09,8.999999E+09]];
    LOCAL CONST Robtarget Tr_meulage_motif_1_300 := [[-78.0860859375,45.72943359375,50.82884765625],[0.376363228761976,-0.369466106511504,0.595187364718739,-0.60629820802494],[0,0,0,0],[8.999999E+09,8.999999E+09,8.999999E+09,8.999999E+09,8.999999E+09,8.999999E+09]];
    LOCAL CONST Robtarget Tr_meulage_motif_1_301 := [[-78.521765625,44.8293359375,50.8288515625],[0.376363228761976,-0.369466106511504,0.595187364718739,-0.60629820802494],[0,0,0,0],[8.999999E+09,8.999999E+09,8.999999E+09,8.999999E+09,8.999999E+09,8.999999E+09]];
    LOCAL CONST Robtarget Tr_meulage_motif_1_302 := [[-78.957453125,43.929234375,50.82885546875],[0.376363228761976,-0.369466106511504,0.595187364718739,-0.60629820802494],[0,0,0,0],[8.999999E+09,8.999999E+09,8.999999E+09,8.999999E+09,8.999999E+09,8.999999E+09]];
    LOCAL CONST Robtarget Tr_meulage_motif_1_303 := [[-79.3931328125,43.02913671875,50.828859375],[0.376363228761976,-0.369466106511504,0.595187364718739,-0.60629820802494],[0,0,0,0],[8.999999E+09,8.999999E+09,8.999999E+09,8.999999E+09,8.999999E+09,8.999999E+09]];
    LOCAL CONST Robtarget Tr_meulage_motif_1_304 := [[-79.8288203125,42.12903515625,50.82886328125],[0.376363228761976,-0.369466106511504,0.595187364718739,-0.60629820802494],[0,0,0,0],[8.999999E+09,8.999999E+09,8.999999E+09,8.999999E+09,8.999999E+09,8.999999E+09]];
    LOCAL CONST Robtarget Tr_meulage_motif_1_305 := [[-80.2645078125,41.2289375,50.8288671875],[0.376363228761976,-0.369466106511504,0.595187364718739,-0.60629820802494],[0,0,0,0],[8.999999E+09,8.999999E+09,8.999999E+09,8.999999E+09,8.999999E+09,8.999999E+09]];
    LOCAL CONST Robtarget Tr_meulage_motif_1_306 := [[-80.7001875,40.3288359375,50.8288671875],[0.376363228761976,-0.369466106511504,0.595187364718739,-0.60629820802494],[0,0,0,0],[8.999999E+09,8.999999E+09,8.999999E+09,8.999999E+09,8.999999E+09,8.999999E+09]];
    LOCAL CONST Robtarget Tr_meulage_motif_1_307 := [[-81.135875,39.42873828125,50.82887109375],[0.376363228761976,-0.369466106511504,0.595187364718739,-0.60629820802494],[0,0,0,0],[8.999999E+09,8.999999E+09,8.999999E+09,8.999999E+09,8.999999E+09,8.999999E+09]];
    LOCAL CONST Robtarget Tr_meulage_motif_1_308 := [[-81.5715546875,38.52863671875,50.828875],[0.376363228761976,-0.369466106511504,0.595187364718739,-0.60629820802494],[0,0,0,0],[8.999999E+09,8.999999E+09,8.999999E+09,8.999999E+09,8.999999E+09,8.999999E+09]];
    LOCAL CONST Robtarget Tr_meulage_motif_1_309 := [[-82.0072421875,37.6285390625,50.82887890625],[0.376363228761976,-0.369466106511504,0.595187364718739,-0.60629820802494],[0,0,0,0],[8.999999E+09,8.999999E+09,8.999999E+09,8.999999E+09,8.999999E+09,8.999999E+09]];
    LOCAL CONST Robtarget Tr_meulage_motif_1_310 := [[-82.4429296875,36.7284375,50.8288828125],[0.376363228761976,-0.369466106511504,0.595187364718739,-0.60629820802494],[0,0,0,0],[8.999999E+09,8.999999E+09,8.999999E+09,8.999999E+09,8.999999E+09,8.999999E+09]];
    LOCAL CONST Robtarget Tr_meulage_motif_1_311 := [[-82.878609375,35.82833984375,50.82888671875],[0.376363228761976,-0.369466106511504,0.595187364718739,-0.60629820802494],[0,0,0,0],[8.999999E+09,8.999999E+09,8.999999E+09,8.999999E+09,8.999999E+09,8.999999E+09]];
    LOCAL CONST Robtarget Tr_meulage_motif_1_312 := [[-83.314296875,34.92823828125,50.828890625],[0.376363228761976,-0.369466106511504,0.595187364718739,-0.60629820802494],[0,0,0,0],[8.999999E+09,8.999999E+09,8.999999E+09,8.999999E+09,8.999999E+09,8.999999E+09]];
    LOCAL CONST Robtarget Tr_meulage_motif_1_313 := [[-83.7499765625,34.028140625,50.828890625],[0.376363228761976,-0.369466106511504,0.595187364718739,-0.60629820802494],[0,0,0,0],[8.999999E+09,8.999999E+09,8.999999E+09,8.999999E+09,8.999999E+09,8.999999E+09]];
    LOCAL CONST Robtarget Tr_meulage_motif_1_314 := [[-84.1856640625,33.12804296875,50.82889453125],[0.376363228761976,-0.369466106511504,0.595187364718739,-0.60629820802494],[0,0,0,0],[8.999999E+09,8.999999E+09,8.999999E+09,8.999999E+09,8.999999E+09,8.999999E+09]];
    LOCAL CONST Robtarget Tr_meulage_motif_1_315 := [[-84.6213515625,32.22794140625,50.8288984375],[0.376363228761976,-0.369466106511504,0.595187364718739,-0.60629820802494],[0,0,0,0],[8.999999E+09,8.999999E+09,8.999999E+09,8.999999E+09,8.999999E+09,8.999999E+09]];
    LOCAL CONST Robtarget Tr_meulage_motif_1_316 := [[-85.05703125,31.327841796875,50.82890234375],[0.376363228761976,-0.369466106511504,0.595187364718739,-0.60629820802494],[0,0,0,0],[8.999999E+09,8.999999E+09,8.999999E+09,8.999999E+09,8.999999E+09,8.999999E+09]];
    LOCAL CONST Robtarget Tr_meulage_motif_1_317 := [[-85.489046875,30.43423046875,50.718296875],[0.376363228761976,-0.369466106511504,0.595187364718739,-0.60629820802494],[0,0,0,0],[8.999999E+09,8.999999E+09,8.999999E+09,8.999999E+09,8.999999E+09,8.999999E+09]];
    LOCAL CONST Robtarget Tr_meulage_motif_1_318 := [[-85.900609375,29.581890625,50.50711328125],[0.376363228761976,-0.369466106511504,0.595187364718739,-0.60629820802494],[0,0,0,0],[8.999999E+09,8.999999E+09,8.999999E+09,8.999999E+09,8.999999E+09,8.999999E+09]];
    LOCAL CONST Robtarget Tr_meulage_motif_1_319 := [[-86.271078125,28.8138515625,50.23529296875],[0.376363228761976,-0.369466106511504,0.595187364718739,-0.60629820802494],[0,0,0,0],[8.999999E+09,8.999999E+09,8.999999E+09,8.999999E+09,8.999999E+09,8.999999E+09]];
    LOCAL CONST Robtarget Tr_meulage_motif_1_320 := [[-86.59675,28.13831640625,49.959359375],[0.376363228761976,-0.369466106511504,0.595187364718739,-0.60629820802494],[0,0,0,0],[8.999999E+09,8.999999E+09,8.999999E+09,8.999999E+09,8.999999E+09,8.999999E+09]];
    LOCAL CONST Robtarget Tr_meulage_motif_1_321 := [[-87.07409375,27.14609765625,49.3432421875],[0.376363228761976,-0.369466106511504,0.595187364718739,-0.60629820802494],[0,0,0,0],[8.999999E+09,8.999999E+09,8.999999E+09,8.999999E+09,8.999999E+09,8.999999E+09]];
    LOCAL CONST Robtarget Tr_meulage_motif_1_322 := [[-87.51690625,26.222923828125,48.49561328125],[0.376363228761976,-0.369466106511504,0.595187364718739,-0.60629820802494],[0,0,0,0],[8.999999E+09,8.999999E+09,8.999999E+09,8.999999E+09,8.999999E+09,8.999999E+09]];
    LOCAL CONST Robtarget Tr_meulage_motif_1_323 := [[-87.8822734375,25.45803515625,47.471765625],[0.376363228761976,-0.369466106511504,0.595187364718739,-0.60629820802494],[0,0,0,0],[8.999999E+09,8.999999E+09,8.999999E+09,8.999999E+09,8.999999E+09,8.999999E+09]];
    LOCAL CONST Robtarget Tr_meulage_motif_1_324 := [[-88.0906484375,25.01655859375,46.35554296875],[0.376363228761976,-0.369466106511504,0.595187364718739,-0.60629820802494],[0,0,0,0],[8.999999E+09,8.999999E+09,8.999999E+09,8.999999E+09,8.999999E+09,8.999999E+09]];
    LOCAL CONST Robtarget Tr_meulage_motif_1_325 := [[-88.0997578125,24.990896484375,45.65961328125],[0.376363228761976,-0.369466106511504,0.595187364718739,-0.60629820802494],[0,0,0,0],[8.999999E+09,8.999999E+09,8.999999E+09,8.999999E+09,8.999999E+09,8.999999E+09]];
    LOCAL CONST Robtarget Tr_meulage_motif_1_326 := [[-88.0972109375,24.98966015625,44.99833984375],[0.376363228761976,-0.369466106511504,0.595187364718739,-0.60629820802494],[0,0,0,0],[8.999999E+09,8.999999E+09,8.999999E+09,8.999999E+09,8.999999E+09,8.999999E+09]];
    LOCAL CONST Robtarget Tr_meulage_motif_1_327 := [[-88.07075,25.037818359375,44.337265625],[0.376363228761976,-0.369466106511504,0.595187364718739,-0.60629820802494],[0,0,0,0],[8.999999E+09,8.999999E+09,8.999999E+09,8.999999E+09,8.999999E+09,8.999999E+09]];
    LOCAL CONST Robtarget Tr_meulage_motif_1_328 := [[-87.8494375,25.484203125,43.2355390625],[0.376363228761976,-0.369466106511504,0.595187364718739,-0.60629820802494],[0,0,0,0],[8.999999E+09,8.999999E+09,8.999999E+09,8.999999E+09,8.999999E+09,8.999999E+09]];
    LOCAL CONST Robtarget Tr_meulage_motif_1_329 := [[-87.4723359375,26.253369140625,42.22890625],[0.376363228761976,-0.369466106511504,0.595187364718739,-0.60629820802494],[0,0,0,0],[8.999999E+09,8.999999E+09,8.999999E+09,8.999999E+09,8.999999E+09,8.999999E+09]];
    LOCAL CONST Robtarget Tr_meulage_motif_1_330 := [[-87.0232578125,27.172986328125,41.40005078125],[0.376363228761976,-0.369466106511504,0.595187364718739,-0.60629820802494],[0,0,0,0],[8.999999E+09,8.999999E+09,8.999999E+09,8.999999E+09,8.999999E+09,8.999999E+09]];
    LOCAL CONST Robtarget Tr_meulage_motif_1_331 := [[-86.722375,27.79069921875,41.00428515625],[0.376363228761976,-0.369466106511504,0.595187364718739,-0.60629820802494],[0,0,0,0],[8.999999E+09,8.999999E+09,8.999999E+09,8.999999E+09,8.999999E+09,8.999999E+09]];
    LOCAL CONST Robtarget Tr_meulage_motif_1_332 := [[-86.21590625,28.832244140625,40.5167578125],[0.376363228761976,-0.369466106511504,0.595187364718739,-0.60629820802494],[0,0,0,0],[8.999999E+09,8.999999E+09,8.999999E+09,8.999999E+09,8.999999E+09,8.999999E+09]];
    LOCAL CONST Robtarget Tr_meulage_motif_1_333 := [[-85.8467265625,29.59236328125,40.25264453125],[0.376363228761976,-0.369466106511504,0.595187364718739,-0.60629820802494],[0,0,0,0],[8.999999E+09,8.999999E+09,8.999999E+09,8.999999E+09,8.999999E+09,8.999999E+09]];
    LOCAL CONST Robtarget Tr_meulage_motif_1_334 := [[-85.439875,30.430873046875,40.04816015625],[0.376363228761976,-0.369466106511504,0.595187364718739,-0.60629820802494],[0,0,0,0],[8.999999E+09,8.999999E+09,8.999999E+09,8.999999E+09,8.999999E+09,8.999999E+09]];
    LOCAL CONST Robtarget Tr_meulage_motif_1_335 := [[-85.0118046875,31.314173828125,39.93961328125],[0.376363228761976,-0.369466106511504,0.595187364718739,-0.60629820802494],[0,0,0,0],[8.999999E+09,8.999999E+09,8.999999E+09,8.999999E+09,8.999999E+09,8.999999E+09]];
    LOCAL CONST Robtarget Tr_meulage_motif_1_336 := [[-84.5789375,32.20737109375,39.829],[0.376363228761976,-0.369466106511504,0.595187364718739,-0.60629820802494],[0,0,0,0],[8.999999E+09,8.999999E+09,8.999999E+09,8.999999E+09,8.999999E+09,8.999999E+09]];
    LOCAL CONST Robtarget Tr_meulage_motif_1_337 := [[-84.14325,33.10747265625,39.82899609375],[0.376363228761976,-0.369466106511504,0.595187364718739,-0.60629820802494],[0,0,0,0],[8.999999E+09,8.999999E+09,8.999999E+09,8.999999E+09,8.999999E+09,8.999999E+09]];
    LOCAL CONST Robtarget Tr_meulage_motif_1_338 := [[-83.7075703125,34.0075703125,39.8289921875],[0.376363228761976,-0.369466106511504,0.595187364718739,-0.60629820802494],[0,0,0,0],[8.999999E+09,8.999999E+09,8.999999E+09,8.999999E+09,8.999999E+09,8.999999E+09]];
    LOCAL CONST Robtarget Tr_meulage_motif_1_339 := [[-83.2718828125,34.907671875,39.82898828125],[0.376363228761976,-0.369466106511504,0.595187364718739,-0.60629820802494],[0,0,0,0],[8.999999E+09,8.999999E+09,8.999999E+09,8.999999E+09,8.999999E+09,8.999999E+09]];
    LOCAL CONST Robtarget Tr_meulage_motif_1_340 := [[-82.836203125,35.80776953125,39.828984375],[0.376363228761976,-0.369466106511504,0.595187364718739,-0.60629820802494],[0,0,0,0],[8.999999E+09,8.999999E+09,8.999999E+09,8.999999E+09,8.999999E+09,8.999999E+09]];
    LOCAL CONST Robtarget Tr_meulage_motif_1_341 := [[-82.400515625,36.70787109375,39.828984375],[0.376363228761976,-0.369466106511504,0.595187364718739,-0.60629820802494],[0,0,0,0],[8.999999E+09,8.999999E+09,8.999999E+09,8.999999E+09,8.999999E+09,8.999999E+09]];
    LOCAL CONST Robtarget Tr_meulage_motif_1_342 := [[-81.964828125,37.60796875,39.82898046875],[0.376363228761976,-0.369466106511504,0.595187364718739,-0.60629820802494],[0,0,0,0],[8.999999E+09,8.999999E+09,8.999999E+09,8.999999E+09,8.999999E+09,8.999999E+09]];
    LOCAL CONST Robtarget Tr_meulage_motif_1_343 := [[-81.5291484375,38.5080703125,39.8289765625],[0.376363228761976,-0.369466106511504,0.595187364718739,-0.60629820802494],[0,0,0,0],[8.999999E+09,8.999999E+09,8.999999E+09,8.999999E+09,8.999999E+09,8.999999E+09]];
    LOCAL CONST Robtarget Tr_meulage_motif_1_344 := [[-81.0934609375,39.40816796875,39.82897265625],[0.376363228761976,-0.369466106511504,0.595187364718739,-0.60629820802494],[0,0,0,0],[8.999999E+09,8.999999E+09,8.999999E+09,8.999999E+09,8.999999E+09,8.999999E+09]];
    LOCAL CONST Robtarget Tr_meulage_motif_1_345 := [[-80.65778125,40.30826953125,39.82896875],[0.376363228761976,-0.369466106511504,0.595187364718739,-0.60629820802494],[0,0,0,0],[8.999999E+09,8.999999E+09,8.999999E+09,8.999999E+09,8.999999E+09,8.999999E+09]];
    LOCAL CONST Robtarget Tr_meulage_motif_1_346 := [[-80.22209375,41.2083671875,39.82896484375],[0.376363228761976,-0.369466106511504,0.595187364718739,-0.60629820802494],[0,0,0,0],[8.999999E+09,8.999999E+09,8.999999E+09,8.999999E+09,8.999999E+09,8.999999E+09]];
    LOCAL CONST Robtarget Tr_meulage_motif_1_347 := [[-79.78640625,42.10846875,39.82896484375],[0.376363228761976,-0.369466106511504,0.595187364718739,-0.60629820802494],[0,0,0,0],[8.999999E+09,8.999999E+09,8.999999E+09,8.999999E+09,8.999999E+09,8.999999E+09]];
    LOCAL CONST Robtarget Tr_meulage_motif_1_348 := [[-79.3507265625,43.00856640625,39.8289609375],[0.376363228761976,-0.369466106511504,0.595187364718739,-0.60629820802494],[0,0,0,0],[8.999999E+09,8.999999E+09,8.999999E+09,8.999999E+09,8.999999E+09,8.999999E+09]];
    LOCAL CONST Robtarget Tr_meulage_motif_1_349 := [[-78.9150390625,43.90866796875,39.82895703125],[0.376363228761976,-0.369466106511504,0.595187364718739,-0.60629820802494],[0,0,0,0],[8.999999E+09,8.999999E+09,8.999999E+09,8.999999E+09,8.999999E+09,8.999999E+09]];
    LOCAL CONST Robtarget Tr_meulage_motif_1_350 := [[-78.479359375,44.808765625,39.828953125],[0.376363228761976,-0.369466106511504,0.595187364718739,-0.60629820802494],[0,0,0,0],[8.999999E+09,8.999999E+09,8.999999E+09,8.999999E+09,8.999999E+09,8.999999E+09]];
    LOCAL CONST Robtarget Tr_meulage_motif_1_351 := [[-78.043671875,45.7088671875,39.82894921875],[0.376363228761976,-0.369466106511504,0.595187364718739,-0.60629820802494],[0,0,0,0],[8.999999E+09,8.999999E+09,8.999999E+09,8.999999E+09,8.999999E+09,8.999999E+09]];
    LOCAL CONST Robtarget Tr_meulage_motif_1_352 := [[-77.6079921875,46.60896484375,39.8289453125],[0.376363228761976,-0.369466106511504,0.595187364718739,-0.60629820802494],[0,0,0,0],[8.999999E+09,8.999999E+09,8.999999E+09,8.999999E+09,8.999999E+09,8.999999E+09]];
    LOCAL CONST Robtarget Tr_meulage_motif_1_353 := [[-77.1723046875,47.50906640625,39.82894140625],[0.376363228761976,-0.369466106511504,0.595187364718739,-0.60629820802494],[0,0,0,0],[8.999999E+09,8.999999E+09,8.999999E+09,8.999999E+09,8.999999E+09,8.999999E+09]];
    LOCAL CONST Robtarget Tr_meulage_motif_1_354 := [[-76.7366171875,48.4091640625,39.82894140625],[0.376363228761976,-0.369466106511504,0.595187364718739,-0.60629820802494],[0,0,0,0],[8.999999E+09,8.999999E+09,8.999999E+09,8.999999E+09,8.999999E+09,8.999999E+09]];
    LOCAL CONST Robtarget Tr_meulage_motif_1_355 := [[-76.3009375,49.309265625,39.8289375],[0.376363228761976,-0.369466106511504,0.595187364718739,-0.60629820802494],[0,0,0,0],[8.999999E+09,8.999999E+09,8.999999E+09,8.999999E+09,8.999999E+09,8.999999E+09]];
    LOCAL CONST Robtarget Tr_meulage_motif_1_356 := [[-75.86525,50.20936328125,39.82893359375],[0.376363228761976,-0.369466106511504,0.595187364718739,-0.60629820802494],[0,0,0,0],[8.999999E+09,8.999999E+09,8.999999E+09,8.999999E+09,8.999999E+09,8.999999E+09]];
    LOCAL CONST Robtarget Tr_meulage_motif_1_357 := [[-75.4295703125,51.10946484375,39.8289296875],[0.376363228761976,-0.369466106511504,0.595187364718739,-0.60629820802494],[0,0,0,0],[8.999999E+09,8.999999E+09,8.999999E+09,8.999999E+09,8.999999E+09,8.999999E+09]];
    LOCAL CONST Robtarget Tr_meulage_motif_1_358 := [[-74.9938828125,52.0095625,39.82892578125],[0.376363228761976,-0.369466106511504,0.595187364718739,-0.60629820802494],[0,0,0,0],[8.999999E+09,8.999999E+09,8.999999E+09,8.999999E+09,8.999999E+09,8.999999E+09]];
    LOCAL CONST Robtarget Tr_meulage_motif_1_359 := [[-74.5581953125,52.9096640625,39.828921875],[0.376363228761976,-0.369466106511504,0.595187364718739,-0.60629820802494],[0,0,0,0],[8.999999E+09,8.999999E+09,8.999999E+09,8.999999E+09,8.999999E+09,8.999999E+09]];
    LOCAL CONST Robtarget Tr_meulage_motif_1_360 := [[-74.122515625,53.80976171875,39.82891796875],[0.376363228761976,-0.369466106511504,0.595187364718739,-0.60629820802494],[0,0,0,0],[8.999999E+09,8.999999E+09,8.999999E+09,8.999999E+09,8.999999E+09,8.999999E+09]];
    LOCAL CONST Robtarget Tr_meulage_motif_1_361 := [[-73.686828125,54.709859375,39.82891796875],[0.376363228761976,-0.369466106511504,0.595187364718739,-0.60629820802494],[0,0,0,0],[8.999999E+09,8.999999E+09,8.999999E+09,8.999999E+09,8.999999E+09,8.999999E+09]];
    LOCAL CONST Robtarget Tr_meulage_motif_1_362 := [[-73.2511484375,55.6099609375,39.8289140625],[0.376363228761976,-0.369466106511504,0.595187364718739,-0.60629820802494],[0,0,0,0],[8.999999E+09,8.999999E+09,8.999999E+09,8.999999E+09,8.999999E+09,8.999999E+09]];
    LOCAL CONST Robtarget Tr_meulage_motif_1_363 := [[-72.8154609375,56.51005859375,39.82891015625],[0.376363228761976,-0.369466106511504,0.595187364718739,-0.60629820802494],[0,0,0,0],[8.999999E+09,8.999999E+09,8.999999E+09,8.999999E+09,8.999999E+09,8.999999E+09]];
    LOCAL CONST Robtarget Tr_meulage_motif_1_364 := [[-72.37978125,57.41016015625,39.82890625],[0.376363228761976,-0.369466106511504,0.595187364718739,-0.60629820802494],[0,0,0,0],[8.999999E+09,8.999999E+09,8.999999E+09,8.999999E+09,8.999999E+09,8.999999E+09]];
    LOCAL CONST Robtarget Tr_meulage_motif_1_365 := [[-71.94409375,58.3102578125,39.82890234375],[0.376363228761976,-0.369466106511504,0.595187364718739,-0.60629820802494],[0,0,0,0],[8.999999E+09,8.999999E+09,8.999999E+09,8.999999E+09,8.999999E+09,8.999999E+09]];
    LOCAL CONST Robtarget Tr_meulage_motif_1_366 := [[-71.50840625,59.210359375,39.8288984375],[0.376363228761976,-0.369466106511504,0.595187364718739,-0.60629820802494],[0,0,0,0],[8.999999E+09,8.999999E+09,8.999999E+09,8.999999E+09,8.999999E+09,8.999999E+09]];
    LOCAL CONST Robtarget Tr_meulage_motif_1_367 := [[-71.0727265625,60.11045703125,39.82889453125],[0.376363228761976,-0.369466106511504,0.595187364718739,-0.60629820802494],[0,0,0,0],[8.999999E+09,8.999999E+09,8.999999E+09,8.999999E+09,8.999999E+09,8.999999E+09]];
    LOCAL CONST Robtarget Tr_meulage_motif_1_368 := [[-70.6370390625,61.01055859375,39.82889453125],[0.376363228761976,-0.369466106511504,0.595187364718739,-0.60629820802494],[0,0,0,0],[8.999999E+09,8.999999E+09,8.999999E+09,8.999999E+09,8.999999E+09,8.999999E+09]];
    LOCAL CONST Robtarget Tr_meulage_motif_1_369 := [[-70.201359375,61.91065625,39.828890625],[0.376363228761976,-0.369466106511504,0.595187364718739,-0.60629820802494],[0,0,0,0],[8.999999E+09,8.999999E+09,8.999999E+09,8.999999E+09,8.999999E+09,8.999999E+09]];
    LOCAL CONST Robtarget Tr_meulage_motif_1_370 := [[-69.765671875,62.8107578125,39.82888671875],[0.376363228761976,-0.369466106511504,0.595187364718739,-0.60629820802494],[0,0,0,0],[8.999999E+09,8.999999E+09,8.999999E+09,8.999999E+09,8.999999E+09,8.999999E+09]];
    LOCAL CONST Robtarget Tr_meulage_motif_1_371 := [[-69.329984375,63.71085546875,39.8288828125],[0.376363228761976,-0.369466106511504,0.595187364718739,-0.60629820802494],[0,0,0,0],[8.999999E+09,8.999999E+09,8.999999E+09,8.999999E+09,8.999999E+09,8.999999E+09]];
    LOCAL CONST Robtarget Tr_meulage_motif_1_372 := [[-68.8943046875,64.61095703125,39.82887890625],[0.376363228761976,-0.369466106511504,0.595187364718739,-0.60629820802494],[0,0,0,0],[8.999999E+09,8.999999E+09,8.999999E+09,8.999999E+09,8.999999E+09,8.999999E+09]];
    LOCAL CONST Robtarget Tr_meulage_motif_1_373 := [[-68.4586171875,65.5110546875,39.828875],[0.376363228761976,-0.369466106511504,0.595187364718739,-0.60629820802494],[0,0,0,0],[8.999999E+09,8.999999E+09,8.999999E+09,8.999999E+09,8.999999E+09,8.999999E+09]];
    LOCAL CONST Robtarget Tr_meulage_motif_1_374 := [[-68.0229375,66.41115625,39.82887109375],[0.376363228761976,-0.369466106511504,0.595187364718739,-0.60629820802494],[0,0,0,0],[8.999999E+09,8.999999E+09,8.999999E+09,8.999999E+09,8.999999E+09,8.999999E+09]];
